	{attribute 'TcIecLibraryType'}
	{attribute 'external_name' := 'F_VN_RemapImageToPolarSpaceExp_GUID_737F4948_F24C_BB66_5AD3_96D65275813B'}
	(* Remap an image to polar space. (expert function) *)
	FUNCTION F_VN_RemapImageToPolarSpaceExp : HRESULT
	VAR_INPUT
		ipSrcImage	:	ITcVnImage;	(* Source image *)
		ipDestImage	:	REFERENCE TO ITcVnImage;	(* Destination image (Must not be the same as ipSrcImage! An appropriate destination image will be created if required.) *)
	END_VAR
	VAR_IN_OUT
		aCenter	:	TcVnPoint2_REAL;	(* Center point for the transformation *)
	END_VAR
	VAR_INPUT
		fMaxRadius	:	LREAL;	(* Maximum radius for the transformation (set to 0 for auto select) *)
		eInterpolationType	:	ETcVnInterpolationType;	(* Interpolation type *)
		hrPrev	:	HRESULT;	(* HRESULT indicating the result of previous operations (If SUCCEEDED(hrPrev) equals false, no operation is executed.) *)
	END_VAR

END_FUNCTION

// Functions/Geometric and Coordinate Transformations/F_VN_RemapImageToPolarSpaceExp2

	{attribute 'TcIecLibraryType'}
	{attribute 'external_name' := 'F_VN_RemapImageToPolarSpaceExp2_GUID_881403E3_891A_BA00_4A88_7979161734A7'}
	(* Remap an image to polar space. (expert function) *)
	FUNCTION F_VN_RemapImageToPolarSpaceExp2 : HRESULT
	VAR_INPUT
		ipSrcImage	:	ITcVnImage;	(* Source image *)
		ipDestImage	:	REFERENCE TO ITcVnImage;	(* Destination image (Must not be the same as ipSrcImage! An appropriate destination image will be created if required.) *)
	END_VAR
	VAR_IN_OUT
		aCenter	:	TcVnPoint2_REAL;	(* Center point for the transformation *)
	END_VAR
	VAR_INPUT
		fMaxRadius	:	LREAL;	(* Maximum radius for the transformation (set to 0 for auto select) *)
		eInterpolationType	:	ETcVnInterpolationType;	(* Interpolation type *)
		nDestWidth	:	DINT;	(* Destination image width (set to -1 for source image width, 0 to auto scale to transformed radius, > 0 for a user defined width) *)
		nDestHeight	:	DINT;	(* destination image height (set to -1 for source image height, 0 to auto scale to transformed radius * PI, > 0 for a user defined height) *)
		hrPrev	:	HRESULT;	(* HRESULT indicating the result of previous operations (If SUCCEEDED(hrPrev) equals false, no operation is executed.) *)
	END_VAR

END_FUNCTION

// Functions/Geometric and Coordinate Transformations/F_VN_ResizeImage

	{attribute 'TcIecLibraryType'}
	{attribute 'external_name' := 'F_VN_ResizeImage_GUID_066F6715_FDC4_B7AC_782D_C69A46C5F7F6'}
	(* Resize an image using a specific interpolation type. *)
	FUNCTION F_VN_ResizeImage : HRESULT
	VAR_INPUT
		ipSrcImage	:	ITcVnImage;	(* Source image *)
		ipDestImage	:	REFERENCE TO ITcVnImage;	(* Destination image (An appropriate image will be created if required.) *)
		nWidth	:	UDINT;	(* New width *)
		nHeight	:	UDINT;	(* New height *)
		eInterpolationType	:	ETcVnInterpolationType;	(* Interpolation type *)
		hrPrev	:	HRESULT;	(* HRESULT indicating the result of previous operations (If SUCCEEDED(hrPrev) equals false, no operation is executed.) *)
	END_VAR

END_FUNCTION

// Functions/Geometric and Coordinate Transformations/F_VN_ResizeImageExp

	{attribute 'TcIecLibraryType'}
	{attribute 'external_name' := 'F_VN_ResizeImageExp_GUID_DC68AAF5_744F_B632_6E74_ACED6F5A8BF2'}
	(* Resize an image using a specific interpolation type while maintaining its aspect ratio. (expert function) *)
	FUNCTION F_VN_ResizeImageExp : HRESULT
	VAR_INPUT
		ipSrcImage	:	ITcVnImage;	(* Source image *)
		ipDestImage	:	REFERENCE TO ITcVnImage;	(* Destination image (An appropriate image will be created if required.) *)
		nWidth	:	UDINT;	(* New width *)
		nHeight	:	UDINT;	(* New height *)
		eInterpolationType	:	ETcVnInterpolationType;	(* Interpolation type *)
		ePaddingMode	:	ETcVnPaddingMode;	(* Image padding mode *)
	END_VAR
	VAR_IN_OUT
		aBorderValue	:	TcVnVector4_LREAL;	(* Border value, if TCVN_PM_LETTERBOX is used *)
	END_VAR
	VAR_INPUT
		hrPrev	:	HRESULT;	(* HRESULT indicating the result of previous operations (If SUCCEEDED(hrPrev) equals false, no operation is executed.) *)
	END_VAR

END_FUNCTION

// Functions/Geometric and Coordinate Transformations/F_VN_RotateImage

	{attribute 'TcIecLibraryType'}
	{attribute 'external_name' := 'F_VN_RotateImage_GUID_67B496A2_F6DE_B78D_5711_982305E4D20B'}
	(* Rotate an image by 90, 180, or 270 degrees in clockwise direction. *)
	FUNCTION F_VN_RotateImage : HRESULT
	VAR_INPUT
		ipSrcImage	:	ITcVnImage;	(* Source image *)
		ipDestImage	:	REFERENCE TO ITcVnImage;	(* Destination image (An appropriate image will be created if required.) *)
		eAngle	:	ETcVnRotationAngle;	(* Rotation angle *)
		hrPrev	:	HRESULT;	(* HRESULT indicating the result of previous operations (If SUCCEEDED(hrPrev) equals false, no operation is executed.) *)
	END_VAR

END_FUNCTION

// Functions/Geometric and Coordinate Transformations/F_VN_RotateImageExp

	{attribute 'TcIecLibraryType'}
	{attribute 'external_name' := 'F_VN_RotateImageExp_GUID_493FD631_7649_B0AF_6E53_B79A69B64150'}
	(* Rotate an image by an individual rotation angle in degrees. *)
	FUNCTION F_VN_RotateImageExp : HRESULT
	VAR_INPUT
		ipSrcImage	:	ITcVnImage;	(* Source image *)
		ipDestImage	:	REFERENCE TO ITcVnImage;	(* Destination image (An appropriate image will be created if required.) *)
		fAngleDeg	:	LREAL;	(* Rotation angle in degree (positive: counter-clockwise, negative: clockwise) *)
		bAdjustDestSize	:	BOOL;	(* If true, ipDestImage size is adjusted so that the whole rotated ipSrcImage is contained. Otherwise, ipDestImage size is set to ipSrcImage size. *)
		hrPrev	:	HRESULT;	(* HRESULT indicating the result of previous operations (If SUCCEEDED(hrPrev) equals false, no operation is executed.) *)
	END_VAR

END_FUNCTION

// Functions/Geometric and Coordinate Transformations/F_VN_RotateImageExp2

	{attribute 'TcIecLibraryType'}
	{attribute 'external_name' := 'F_VN_RotateImageExp2_GUID_6EE8673E_D50E_BAEC_65C2_A62D1613988A'}
	(* Rotate an image by an individual rotation angle in degrees. (expert function) *)
	FUNCTION F_VN_RotateImageExp2 : HRESULT
	VAR_INPUT
		ipSrcImage	:	ITcVnImage;	(* Source image *)
		ipDestImage	:	REFERENCE TO ITcVnImage;	(* Destination image (An appropriate image will be created if required.) *)
		fAngleDeg	:	LREAL;	(* Rotation angle in degree (positive: counter-clockwise, negative: clockwise) *)
		bAdjustDestSize	:	BOOL;	(* If true, ipDestImage size is adjusted so that the whole rotated ipSrcImage is contained. Otherwise, ipDestImage size is set to ipSrcImage size. *)
		eInterpolationType	:	ETcVnInterpolationType;	(* Interpolation method *)
		eBorderInterpolation	:	ETcVnBorderInterpolationMethod;	(* Border interpolation method (ISOLATED not supported) *)
	END_VAR
	VAR_IN_OUT
		aBorderValue	:	TcVnVector4_LREAL;	(* Border value, if CONSTANT is used *)
	END_VAR
	VAR_INPUT
		hrPrev	:	HRESULT;	(* HRESULT indicating the result of previous operations (If SUCCEEDED(hrPrev) equals false, no operation is executed.) *)
	END_VAR

END_FUNCTION

// Functions/Geometric and Coordinate Transformations/F_VN_WarpAffineExp

	{attribute 'TcIecLibraryType'}
	{attribute 'external_name' := 'F_VN_WarpAffineExp_GUID_0ED46A98_6634_BCF0_4EEE_5250D0F0F4C5'}
	(* Apply an affine transformation to an image. (expert function) *)
	FUNCTION F_VN_WarpAffineExp : HRESULT
	VAR_INPUT
		ipSrcImage	:	ITcVnImage;	(* Source image *)
		ipDestImage	:	REFERENCE TO ITcVnImage;	(* Destination image (An appropriate image will be created if required.) *)
	END_VAR
	VAR_IN_OUT
		aTransformationMatrix	:	TcVnMatrix2x3_LREAL;	(* Affine transformation matrix *)
	END_VAR
	VAR_INPUT
		nDestWidth	:	UDINT;	(* Width of the destination image *)
		nDestHeight	:	UDINT;	(* Height of the destination image *)
		eInterpolationType	:	ETcVnInterpolationType;	(* Interpolation method *)
		bWarpInverse	:	BOOL;	(* Handle aTransformationMatrix as the inverse transformation *)
		eBorderInterpolation	:	ETcVnBorderInterpolationMethod;	(* Border interpolation method (ISOLATED not supported) *)
		fBorderValue	:	LREAL;	(* Border value, if CONSTANT is used *)
		hrPrev	:	HRESULT;	(* HRESULT indicating the result of previous operations (If SUCCEEDED(hrPrev) equals false, no operation is executed.) *)
	END_VAR

END_FUNCTION

// Functions/Geometric and Coordinate Transformations/F_VN_WarpAffine_Container

	{attribute 'TcIecLibraryType'}
	{attribute 'external_name' := 'F_VN_WarpAffine_Container_GUID_56BD7DA6_1D43_BE4D_7B12_DD5C0D5972CA'}
	(* Apply an affine transformation to a container of 2D points. *)
	FUNCTION F_VN_WarpAffine_Container : HRESULT
	VAR_INPUT
		ipSrcPoints	:	ITcVnContainer;	(* Source points (ContainerType_Vector_TcVnPoint2_DINT or ContainerType_Vector_TcVnPoint2_REAL or ContainerType_Vector_TcVnPoint2_LREAL) *)
		ipDestPoints	:	REFERENCE TO ITcVnContainer;	(* Returns the transformed points (same type ID as ipSrcPoints; Non-zero interface pointers are reused.) *)
	END_VAR
	VAR_IN_OUT
		aTransformationMatrix	:	TcVnMatrix2x3_LREAL;	(* Affine transformation matrix *)
	END_VAR
	VAR_INPUT
		hrPrev	:	HRESULT;	(* HRESULT indicating the result of previous operations (If SUCCEEDED(hrPrev) equals false, no operation is executed.) *)
	END_VAR

END_FUNCTION

// Functions/Geometric and Coordinate Transformations/F_VN_WarpAffine_Point

	{attribute 'TcIecLibraryType'}
	{attribute 'external_name' := 'F_VN_WarpAffine_Point_GUID_E77A0286_2158_BB35_4767_1C578A33A298'}
	(* Apply an affine transformation to a 2D point. *)
	FUNCTION F_VN_WarpAffine_Point : HRESULT
	VAR_IN_OUT
		aSrcPoint	:	TcVnPoint2_LREAL;	(* Source point *)
		aDestPoint	:	TcVnPoint2_LREAL;	(* Destination point *)
		aTransformationMatrix	:	TcVnMatrix2x3_LREAL;	(* Affine transformation matrix *)
	END_VAR
	VAR_INPUT
		hrPrev	:	HRESULT;	(* HRESULT indicating the result of previous operations (If SUCCEEDED(hrPrev) equals false, no operation is executed.) *)
	END_VAR

END_FUNCTION

// Functions/Geometric and Coordinate Transformations/F_VN_WarpAffine_Rectangle

	{attribute 'TcIecLibraryType'}
	{attribute 'external_name' := 'F_VN_WarpAffine_Rectangle_GUID_B71280DA_6C13_B846_4078_31BCF2965F61'}
	(* Use an affine transform to warp a rectangle. *)
	FUNCTION F_VN_WarpAffine_Rectangle : HRESULT
	VAR_INPUT
		nTopLeftX	:	UDINT;	(* x coordinate of the top left corner *)
		nTopLeftY	:	UDINT;	(* y coordinate of the top left corner *)
		nBottomRightX	:	UDINT;	(* x coordinate of the bottom right corner *)
		nBottomRightY	:	UDINT;	(* y coordinate of the bottom right corner *)
		ipDestPoints	:	REFERENCE TO ITcVnContainer;	(* Returns the 4 transformed points (ContainerType_Vector_TcVnPoint2_REAL) *)
	END_VAR
	VAR_IN_OUT
		aTransformationMatrix	:	TcVnMatrix2x3_LREAL;	(* Affine transformation matrix *)
	END_VAR
	VAR_INPUT
		hrPrev	:	HRESULT;	(* HRESULT indicating the result of previous operations (If SUCCEEDED(hrPrev) equals false, no operation is executed.) *)
	END_VAR

END_FUNCTION

// Functions/Geometric and Coordinate Transformations/F_VN_WarpPerspective

	{attribute 'TcIecLibraryType'}
	{attribute 'external_name' := 'F_VN_WarpPerspective_GUID_11483E27_169B_BD3A_571C_EBB12C538839'}
	(* Apply a perspective transformation to an image. *)
	FUNCTION F_VN_WarpPerspective : HRESULT
	VAR_INPUT
		ipSrcImage	:	ITcVnImage;	(* Source image *)
		ipDestImage	:	REFERENCE TO ITcVnImage;	(* Destination image (An appropriate image will be created if required.) *)
	END_VAR
	VAR_IN_OUT
		aTransformationMatrix	:	TcVnMatrix3x3_LREAL;	(* Perspective transformation matrix *)
	END_VAR
	VAR_INPUT
		hrPrev	:	HRESULT;	(* HRESULT indicating the result of previous operations (If SUCCEEDED(hrPrev) equals false, no operation is executed.) *)
	END_VAR

END_FUNCTION

// Functions/Geometric and Coordinate Transformations/F_VN_WarpPerspective_Container

	{attribute 'TcIecLibraryType'}
	{attribute 'external_name' := 'F_VN_WarpPerspective_Container_GUID_1A9D55A3_310D_B2CA_7120_BA66C8FDA0DB'}
	(* Apply a perspective transformation to a container of 2D points. *)
	FUNCTION F_VN_WarpPerspective_Container : HRESULT
	VAR_INPUT
		ipSrcPoints	:	ITcVnContainer;	(* Source points (ContainerType_Vector_TcVnPoint2_DINT or ContainerType_Vector_TcVnPoint2_REAL or ContainerType_Vector_TcVnPoint2_LREAL) *)
		ipDestPoints	:	REFERENCE TO ITcVnContainer;	(* Returns the transformed points (same type ID as ipSrcPoints; Non-zero interface pointers are reused.) *)
	END_VAR
	VAR_IN_OUT
		aTransformationMatrix	:	TcVnMatrix3x3_LREAL;	(* Perspective transformation matrix *)
	END_VAR
	VAR_INPUT
		hrPrev	:	HRESULT;	(* HRESULT indicating the result of previous operations (If SUCCEEDED(hrPrev) equals false, no operation is executed.) *)
	END_VAR

END_FUNCTION

// Functions/Geometric and Coordinate Transformations/F_VN_WarpPerspectiveExp

	{attribute 'TcIecLibraryType'}
	{attribute 'external_name' := 'F_VN_WarpPerspectiveExp_GUID_EA1E1C8D_C6BD_B82F_4255_245E461C95D7'}
	(* Apply a perspective transformation to an image. (expert function) *)
	FUNCTION F_VN_WarpPerspectiveExp : HRESULT
	VAR_INPUT
		ipSrcImage	:	ITcVnImage;	(* Source image *)
		ipDestImage	:	REFERENCE TO ITcVnImage;	(* Destination image (An appropriate image will be created if required.) *)
	END_VAR
	VAR_IN_OUT
		aTransformationMatrix	:	TcVnMatrix3x3_LREAL;	(* Perspective transformation matrix *)
	END_VAR
	VAR_INPUT
		nDestWidth	:	UDINT;	(* Width of the destination image *)
		nDestHeight	:	UDINT;	(* Height of the destination image *)
		eInterpolationType	:	ETcVnInterpolationType;	(* Interpolation method *)
		bWarpInverse	:	BOOL;	(* Handle aTransformationMatrix as the inverse transformation *)
		eBorderInterpolation	:	ETcVnBorderInterpolationMethod;	(* Border interpolation method (ISOLATED not supported) *)
		fBorderValue	:	LREAL;	(* Border value, if CONSTANT is used *)
		hrPrev	:	HRESULT;	(* HRESULT indicating the result of previous operations (If SUCCEEDED(hrPrev) equals false, no operation is executed.) *)
	END_VAR

END_FUNCTION

// Functions/Geometric and Coordinate Transformations/F_VN_WarpPerspective_Point

	{attribute 'TcIecLibraryType'}
	{attribute 'external_name' := 'F_VN_WarpPerspective_Point_GUID_E1C023CB_EEE0_BA8C_5D66_DED344D33911'}
	(* Apply a perspective transformation to a 2D point. *)
	FUNCTION F_VN_WarpPerspective_Point : HRESULT
	VAR_IN_OUT
		aSrcPoint	:	TcVnPoint2_LREAL;	(* Source point *)
		aDestPoint	:	TcVnPoint2_LREAL;	(* Destination point *)
		aTransformationMatrix	:	TcVnMatrix3x3_LREAL;	(* Perspective transformation matrix *)
	END_VAR
	VAR_INPUT
		hrPrev	:	HRESULT;	(* HRESULT indicating the result of previous operations (If SUCCEEDED(hrPrev) equals false, no operation is executed.) *)
	END_VAR

END_FUNCTION

// Functions/Geometric and Coordinate Transformations/F_VN_WarpPerspective_Rectangle

	{attribute 'TcIecLibraryType'}
	{attribute 'external_name' := 'F_VN_WarpPerspective_Rectangle_GUID_17AD1D40_0ED8_BEB6_46C5_9351EA5858B8'}
	(* Use a perspective transform to warp a rectangle. *)
	FUNCTION F_VN_WarpPerspective_Rectangle : HRESULT
	VAR_INPUT
		nTopLeftX	:	UDINT;	(* x coordinate of the top left corner *)
		nTopLeftY	:	UDINT;	(* y coordinate of the top left corner *)
		nBottomRightX	:	UDINT;	(* x coordinate of the bottom right corner *)
		nBottomRightY	:	UDINT;	(* y coordinate of the bottom right corner *)
		ipDestPoints	:	REFERENCE TO ITcVnContainer;	(* Returns the 4 transformed points (ContainerType_Vector_TcVnPoint2_REAL) *)
	END_VAR
	VAR_IN_OUT
		aTransformationMatrix	:	TcVnMatrix3x3_LREAL;	(* Perspective transformation matrix *)
	END_VAR
	VAR_INPUT
		hrPrev	:	HRESULT;	(* HRESULT indicating the result of previous operations (If SUCCEEDED(hrPrev) equals false, no operation is executed.) *)
	END_VAR

END_FUNCTION

// Functions/Image Color and Contrast Processing/F_VN_ApplyColorMap

	{attribute 'TcIecLibraryType'}
	{attribute 'external_name' := 'F_VN_ApplyColorMap_GUID_816CD833_E52B_BFA9_5F37_7447DD2AD7D0'}
	(* Apply a color map to a gray-level image. *)
	FUNCTION F_VN_ApplyColorMap : HRESULT
	VAR_INPUT
		ipSrcImage	:	ITcVnImage;	(* Source image (TCVN_ET_USINT or TCVN_ET_UINT, 1 channel) *)
		ipDestImage	:	REFERENCE TO ITcVnImage;	(* Returns the colored image (TCVN_ET_USINT, 3 channel. An appropriate image will be created if required.) *)
		ipColorMap	:	ITcVnContainer;	(* Color map to be applied to ipSrcImage (ContainerType_Vector_TcVnVector3_REAL with 256 or 65536 elements, dependent on ipSrcImage type). Can be either custom or created with F_VN_GenerateColorMap. *)
		hrPrev	:	HRESULT;	(* HRESULT indicating the result of previous operations (If SUCCEEDED(hrPrev) equals false, no operation is executed.) *)
	END_VAR

END_FUNCTION

// Functions/Image Color and Contrast Processing/F_VN_GenerateColorMap

	{attribute 'TcIecLibraryType'}
	{attribute 'external_name' := 'F_VN_GenerateColorMap_GUID_9FBF6773_DCEB_B6C6_7464_04D1C3DACD57'}
	(* Generates a pre-defined color map. *)
	FUNCTION F_VN_GenerateColorMap : HRESULT
	VAR_INPUT
		ipColorMap	:	REFERENCE TO ITcVnContainer;	(* Returns the color map (ContainerType_Vector_TcVnVector3_REAL with 256 or 65536 elements) *)
		eColorMap	:	ETcVnColorMap;	(* Selects a color map (similar to GNU Octave/MATLAB types) *)
		eColorMapSize	:	ETcVnColorMapSize;	(* Defines how many elements the generated color map should have *)
		hrPrev	:	HRESULT;	(* HRESULT indicating the result of previous operations (If SUCCEEDED(hrPrev) equals false, no operation is executed.) *)
	END_VAR

END_FUNCTION

// Functions/Image Color and Contrast Processing/F_VN_ApplyLut

	{attribute 'TcIecLibraryType'}
	{attribute 'external_name' := 'F_VN_ApplyLut_GUID_83DE5545_7633_BB82_50E7_190747D5A6CE'}
	(* Apply a lookup table to an image to manipulate its colors. *)
	FUNCTION F_VN_ApplyLut : HRESULT
	VAR_INPUT
		ipSrcImage	:	ITcVnImage;	(* Source image (1-4 channels of 8 or 16 bit types SINT, USINT, INT, UINT) *)
		ipDestImage	:	REFERENCE TO ITcVnImage;	(* Returns the result image (same size, type and channels as ipSrcImage. An appropriate image will be created if required.) *)
		ipLut	:	ITcVnContainer;	(* Lookup table with elements matching ipSrcImage type and either 256 (8 bit images) or 65536 (16 bit images) elements. E.g. ContainerType_Vector_USINT for 1-4 channel USINT image (in this case, the same lookup values are used for each channel) or ContainerType_Vector_TcVnVector3_USINT for a 3 channel USINT image (in this case, each channel uses an individual lookup value).
						 *)
		hrPrev	:	HRESULT;	(* HRESULT indicating the result of previous operations (If SUCCEEDED(hrPrev) equals false, no operation is executed.) *)
	END_VAR

END_FUNCTION

// Functions/Image Color and Contrast Processing/F_VN_Clahe

	{attribute 'TcIecLibraryType'}
	{attribute 'external_name' := 'F_VN_Clahe_GUID_B13FB575_AC4E_B224_67EF_0C730B48FF00'}
	(* Apply Constrast Limited Adaptive Histogram Equalization. This applies local histogram equalization to individual tiles. *)
	FUNCTION F_VN_Clahe : HRESULT
	VAR_INPUT
		ipSrcImage	:	ITcVnImage;	(* Source image (TCVN_ET_USINT or TCVN_ET_UINT, 1 channel) *)
		ipDestImage	:	REFERENCE TO ITcVnImage;	(* Returns the resulting image (An appropriate image will be created if required.) *)
		hrPrev	:	HRESULT;	(* HRESULT indicating the result of previous operations (If SUCCEEDED(hrPrev) equals false, no operation is executed.) *)
	END_VAR

END_FUNCTION

// Functions/Image Color and Contrast Processing/F_VN_ClaheExp

	{attribute 'TcIecLibraryType'}
	{attribute 'external_name' := 'F_VN_ClaheExp_GUID_0B0380D7_C764_B242_5B93_4C54EB94AC2E'}
	(* Apply Constrast Limited Adaptive Histogram Equalization. This applies local histogram equalization to individual tiles. (expert function) *)
	FUNCTION F_VN_ClaheExp : HRESULT
	VAR_INPUT
		ipSrcImage	:	ITcVnImage;	(* Source image (TCVN_ET_USINT or TCVN_ET_UINT, 1 channel) *)
		ipDestImage	:	REFERENCE TO ITcVnImage;	(* Returns the resulting image (An appropriate image will be created if required.) *)
		fClipLimit	:	LREAL;	(* Threshold for contrast limit (set to <= 0 to disable clipping) *)
		nTilesX	:	UDINT;	(* Number of tiles in x direction *)
		nTilesY	:	UDINT;	(* Number of tiles in y direction *)
		hrPrev	:	HRESULT;	(* HRESULT indicating the result of previous operations (If SUCCEEDED(hrPrev) equals false, no operation is executed.) *)
	END_VAR

END_FUNCTION

// Functions/Image Color and Contrast Processing/F_VN_ConvertColorSpace

	{attribute 'TcIecLibraryType'}
	{attribute 'external_name' := 'F_VN_ConvertColorSpace_GUID_E785C056_EC91_BB5D_5362_B1636F1941D4'}
	(* Convert image from one color space to another. *)
	FUNCTION F_VN_ConvertColorSpace : HRESULT
	VAR_INPUT
		ipSrcImage	:	ITcVnImage;	(* Source image *)
		ipDestImage	:	REFERENCE TO ITcVnImage;	(* Destination image (An appropriate destination image will be created if required.) *)
		eTransform	:	ETcVnColorSpaceTransform;	(* Transforms to be applied *)
		hrPrev	:	HRESULT;	(* HRESULT indicating the result of previous operations (If SUCCEEDED(hrPrev) equals false, no operation is executed.) *)
	END_VAR

END_FUNCTION

// Functions/Image Color and Contrast Processing/F_VN_GenerateCustomColorMap

	{attribute 'TcIecLibraryType'}
	{attribute 'external_name' := 'F_VN_GenerateCustomColorMap_GUID_FB8B79DD_6786_B6EC_65F8_CD6C6281E850'}
	(* Generate a custom color map by interpolating between user defined colors (equally distributed, linear for each channel). *)
	FUNCTION F_VN_GenerateCustomColorMap : HRESULT
	VAR_INPUT
		ipColorMap	:	REFERENCE TO ITcVnContainer;	(* Returns the color map (ContainerType_Vector_TcVnVector3_REAL with 256 or 65536 elements) *)
		ipInitialColors	:	ITcVnContainer;	(* User defined colors (ContainerType_Vector_TcVnVector3_REAL, at least 2 elements) *)
		eColorMapSize	:	ETcVnColorMapSize;	(* Defines how many elements the generated color map should have *)
		hrPrev	:	HRESULT;	(* HRESULT indicating the result of previous operations (If SUCCEEDED(hrPrev) equals false, no operation is executed.) *)
	END_VAR

END_FUNCTION

// Functions/Image Color and Contrast Processing/F_VN_Histogram

	{attribute 'TcIecLibraryType'}
	{attribute 'external_name' := 'F_VN_Histogram_GUID_97CA8631_C257_B622_4550_DD2D53C6AEF0'}
	(* Calculate the (multi-channel) histogram of an image. *)
	FUNCTION F_VN_Histogram : HRESULT
	VAR_INPUT
		ipSrcImage	:	ITcVnImage;	(* Source image *)
		ipDestHistogram	:	REFERENCE TO ITcVnContainer;	(* Returns a container with a multi-channel histogram, where every channel is represented as a vector of UDINT (ContainerType_Vector_Vector_UDINT. Non-zero interface pointers are reused.) *)
		hrPrev	:	HRESULT;	(* HRESULT indicating the result of previous operations (If SUCCEEDED(hrPrev) equals false, no operation is executed.) *)
	END_VAR

END_FUNCTION

// Functions/Image Color and Contrast Processing/F_VN_HistogramExp

	{attribute 'TcIecLibraryType'}
	{attribute 'external_name' := 'F_VN_HistogramExp_GUID_1CE0E788_2C38_B155_6387_B008436334A8'}
	(* Calculate the (multi-channel) histogram of an image. (expert function) *)
	FUNCTION F_VN_HistogramExp : HRESULT
	VAR_INPUT
		ipSrcImage	:	ITcVnImage;	(* Source image *)
		ipDestHistogram	:	REFERENCE TO ITcVnContainer;	(* Returns a container with a multi-channel histogram, where every channel is represented as a vector of UDINT (ContainerType_Vector_Vector_UDINT. Non-zero interface pointers are reused.) *)
	END_VAR
	VAR_IN_OUT
		nBins	:	UDINT;	(* Desired number of bins or 0 to keep the default for the corresponding image format (in) and default number of bins (out) *)
		fLowerBound	:	LREAL;	(* Lower (inclusive) boundary of the 0-th histogram bin (in), or receive the default if fLowerBound AND fUpperBound are set to 0 (out) *)
		fUpperBound	:	LREAL;	(* Upper (exclusive) boundary of the last histogram bin nBins-1 (in), or receive the default if fLowerBound AND fUpperBound are set to 0 (out) *)
	END_VAR
	VAR_INPUT
		ipMask	:	ITcVnImage;	(* Source image mask (TCVN_ET_USINT, 1 channel. Mask is optional, set to 0 if not required.) *)
		hrPrev	:	HRESULT;	(* HRESULT indicating the result of previous operations (If SUCCEEDED(hrPrev) equals false, no operation is executed.) *)
	END_VAR

END_FUNCTION

// Functions/Image Color and Contrast Processing/F_VN_HistogramEqualization

	{attribute 'TcIecLibraryType'}
	{attribute 'external_name' := 'F_VN_HistogramEqualization_GUID_3A0A3442_60A5_B388_5E3C_3DBC771CEFC5'}
	(* Equalize the histogram of a grayscale or rgb image, which normalizes the brightness and improves the contrast. *)
	FUNCTION F_VN_HistogramEqualization : HRESULT
	VAR_INPUT
		ipSrcImage	:	ITcVnImage;	(* Source image (USINT) *)
		ipDestImage	:	REFERENCE TO ITcVnImage;	(* Destination image (An appropriate destination image will be created if required.) *)
		hrPrev	:	HRESULT;	(* HRESULT indicating the result of previous operations (If SUCCEEDED(hrPrev) equals false, no operation is executed.) *)
	END_VAR

END_FUNCTION

// Functions/Image Color and Contrast Processing/F_VN_HistogramEqualizationExp

	{attribute 'TcIecLibraryType'}
	{attribute 'external_name' := 'F_VN_HistogramEqualizationExp_GUID_5019ED08_9A6E_BC80_7357_425A106A22F3'}
	(* Equalize the histogram of a grayscale or color image, which normalizes the brightness and improves the contrast. (expert function) 
	The channel index that should be equalized has to be specified (-1 expects a RGB image, converts it to YCbCr, equalizes the Y channel and converts the image back to RGB).  *)
	FUNCTION F_VN_HistogramEqualizationExp : HRESULT
	VAR_INPUT
		ipSrcImage	:	ITcVnImage;	(* Source image (USINT) *)
		ipDestImage	:	REFERENCE TO ITcVnImage;	(* Destination image (An appropriate destination image will be created if required.) *)
		nChannelIdx	:	INT;	(* Index of the image channel that should be equalized (-1 expects a RGB image, converts it to YCbCr, equalizes the Y channel and converts the image back to RGB) *)
		hrPrev	:	HRESULT;	(* HRESULT indicating the result of previous operations (If SUCCEEDED(hrPrev) equals false, no operation is executed.) *)
	END_VAR

END_FUNCTION

// Functions/Image Color and Contrast Processing/F_VN_InvertImageColor

	{attribute 'TcIecLibraryType'}
	{attribute 'external_name' := 'F_VN_InvertImageColor_GUID_E911183A_FFD5_BC4C_5076_3C639D48FDD8'}
	(* Invert the color of an image.
          For signed integer or negative floating point values, only the signs will be switched.
          If the image contains only positive floating point values, each pixel value is subtracted from the maximum available pixel value (or 1.0, whatever is higher). *)
	FUNCTION F_VN_InvertImageColor : HRESULT
	VAR_INPUT
		ipSrcImage	:	ITcVnImage;	(* Source image *)
		ipDestImage	:	REFERENCE TO ITcVnImage;	(* Destination image (An appropriate image will be created if required.) *)
		hrPrev	:	HRESULT;	(* HRESULT indicating the result of previous operations (If SUCCEEDED(hrPrev) equals false, no operation is executed.) *)
	END_VAR

END_FUNCTION

// Functions/Image Color and Contrast Processing/F_VN_InvertImageColorExp

	{attribute 'TcIecLibraryType'}
	{attribute 'external_name' := 'F_VN_InvertImageColorExp_GUID_06670B20_9EED_BCE6_6339_608C38CC3C14'}
	(* Invert the color of an image. (expert function)
          For signed integer or negative floating point values, only the signs will be switched.
          If the image contains only positive floating point values, each pixel value is subtracted from the maximum available pixel value (or 1.0, whatever is higher). *)
	FUNCTION F_VN_InvertImageColorExp : HRESULT
	VAR_INPUT
		ipSrcImage	:	ITcVnImage;	(* Source image *)
		ipDestImage	:	REFERENCE TO ITcVnImage;	(* Destination image (An appropriate image will be created if required.) *)
		fMaxValue	:	LREAL;	(* Maximum pixel value (e.g. if a 16 bit image contains 12 bit values). -1 means the default values are used. *)
		hrPrev	:	HRESULT;	(* HRESULT indicating the result of previous operations (If SUCCEEDED(hrPrev) equals false, no operation is executed.) *)
	END_VAR

END_FUNCTION

// Functions/Image Color and Contrast Processing/F_VN_NormalizeImage

	{attribute 'TcIecLibraryType'}
	{attribute 'external_name' := 'F_VN_NormalizeImage_GUID_DF64614F_1E7D_BDE6_6A3D_02BF884DF440'}
	(* Normalize an image regarding its value range (e.g. stretch pixel values [50..150] to full range [0..255]). *)
	FUNCTION F_VN_NormalizeImage : HRESULT
	VAR_INPUT
		ipSrcImage	:	ITcVnImage;	(* Source image *)
		ipDestImage	:	REFERENCE TO ITcVnImage;	(* Destination image (An appropriate destination image will be created if required.) *)
		hrPrev	:	HRESULT;	(* HRESULT indicating the result of previous operations (If SUCCEEDED(hrPrev) equals false, no operation is executed.) *)
	END_VAR

END_FUNCTION

// Functions/Image Color and Contrast Processing/F_VN_NormalizeImageExp

	{attribute 'TcIecLibraryType'}
	{attribute 'external_name' := 'F_VN_NormalizeImageExp_GUID_278826A3_5B31_B86C_4F2C_A4B2EC762E0C'}
	(* Normalize an image regarding its value range (e.g. stretch pixel values [50..150] to full range [0..255]) or scale the values regarding a specific normalization (e.g. L2-norm). (expert function) *)
	FUNCTION F_VN_NormalizeImageExp : HRESULT
	VAR_INPUT
		ipSrcImage	:	ITcVnImage;	(* Source image *)
		ipDestImage	:	REFERENCE TO ITcVnImage;	(* Destination image (An appropriate destination image will be created if required.) *)
		fAlpha	:	LREAL;	(* Lower range boundary (in case of normalizing the value range) or value to normalize to (||ipDestImage|| = fAlpha) *)
		fBeta	:	LREAL;	(* Upper range boundary (in case of normalizing the value range) *)
		eNormType	:	ETcVnNormalizationType;	(* Normalization type (only INF, L1, L2 or MINMAX) *)
		eDestType	:	ETcVnElementType;	(* Destination image depth (usually SAME_AS_SOURCE) *)
		ipMask	:	ITcVnImage;	(* Mask to restrict the normalization to specific pixel positions (set 0 to normalize the whole image) *)
		hrPrev	:	HRESULT;	(* HRESULT indicating the result of previous operations (If SUCCEEDED(hrPrev) equals false, no operation is executed.) *)
	END_VAR

END_FUNCTION

// Functions/Image Color and Contrast Processing/F_VN_NormalizeImageForDisplay

	{attribute 'TcIecLibraryType'}
	{attribute 'external_name' := 'F_VN_NormalizeImageForDisplay_GUID_849482CC_D1BF_B1BB_6D8E_6AC161F307DE'}
	(* Normalize an image for display, i.e. scale it to the full value range of the underlying data type (-1 to 1 for floating point). *)
	FUNCTION F_VN_NormalizeImageForDisplay : HRESULT
	VAR_INPUT
		ipSrcImage	:	ITcVnImage;	(* Source image *)
		ipDestImage	:	REFERENCE TO ITcVnImage;	(* Destination image (An appropriate destination image will be created if required.) *)
		eSignedNormalization	:	ETcVnSignedNormalization;	(* Option for normalizing signed values *)
		hrPrev	:	HRESULT;	(* HRESULT indicating the result of previous operations (If SUCCEEDED(hrPrev) equals false, no operation is executed.) *)
	END_VAR

END_FUNCTION

// Functions/Image Color and Contrast Processing/F_VN_ReferenceColorSimilarity_ITcVnColorModel

	{attribute 'TcIecLibraryType'}
	{attribute 'external_name' := 'F_VN_ReferenceColorSimilarity_ITcVnColorModel_GUID_F4B25797_7917_B8FC_5558_54102443F353'}
	(* Computes the similarity to a reference color model for each pixel in the source image. *)
	FUNCTION F_VN_ReferenceColorSimilarity_ITcVnColorModel : HRESULT
	VAR_INPUT
		ipSrcImage	:	ITcVnImage;	(* RGB source image (USINT, 3 channels) *)
		ipDestImage	:	REFERENCE TO ITcVnImage;	(* Returns the similarity to ipColorModel for each pixel in ipSrcImage (USINT, 1 channel. An appropriate destination image will be created if required.) *)
		ipColorModel	:	ITcVnColorModel;	(* Color model *)
		hrPrev	:	HRESULT;	(* HRESULT indicating the result of previous operations (If SUCCEEDED(hrPrev) equals false, no operation is executed.) *)
	END_VAR

END_FUNCTION

// Interfaces/Machine Learning/ITcVnColorModel

	(* Interface to train and classify an image color. *)
	{attribute 'c++_compatible'}
	{attribute 'vtable_order' := 'TrainImageColor;ClassifyImageColor'}
	INTERFACE ITcVnColorModel EXTENDS ITcVnMlModel


(* Train the color of the provided image. *)
	{attribute 'c++_compatible'}
	{attribute 'minimal_input_size' := '4'}
	{attribute 'pack_mode' := '4'}
	METHOD TrainImageColor : HRESULT
	VAR_INPUT
		ipSrcImage : ITcVnImage;
		nDifferentColors : UDINT;
		ipMask : ITcVnImage;
		nSkipPixels : UDINT;
	END_VAR
END_METHOD


(* Compute the similarity of each image pixel to the trained reference color. *)
	{attribute 'c++_compatible'}
	{attribute 'minimal_input_size' := '4'}
	{attribute 'pack_mode' := '4'}
	METHOD ClassifyImageColor : HRESULT
	VAR_INPUT
		ipSrcImage : ITcVnImage;
		pipDestImage : POINTER TO ITcVnImage;
		fVariance : REAL;
		fLuminanceWeight : REAL;
	END_VAR
END_METHOD

END_INTERFACE

// Functions/Image Color and Contrast Processing/F_VN_ReferenceColorSimilarityExp_ITcVnColorModel

	{attribute 'TcIecLibraryType'}
	{attribute 'external_name' := 'F_VN_ReferenceColorSimilarityExp_ITcVnColorModel_GUID_F0AE672C_F0E6_B94B_7FE1_8AB59959B227'}
	(* Computes the similarity to a reference color model for each pixel in the source image. (expert function) *)
	FUNCTION F_VN_ReferenceColorSimilarityExp_ITcVnColorModel : HRESULT
	VAR_INPUT
		ipSrcImage	:	ITcVnImage;	(* RGB source image (USINT, 3 channels) *)
		ipDestImage	:	REFERENCE TO ITcVnImage;	(* Returns the similarity to ipColorModel for each pixel in ipSrcImage (USINT, 1 channel. An appropriate destination image will be created if required.) *)
		ipColorModel	:	ITcVnColorModel;	(* Color model *)
		fVariance	:	REAL;	(* Allowed color variance (0.1 - 0.3 might be a good start to try) *)
		fLuminanceWeight	:	REAL;	(* Weight the impact of the luminance ([0..1], e.g. set to 0 to be more resistant to unequal illumination, but might be required to differentiate between some colors. Ignored if ipColorModel is of type RGB.) *)
		hrPrev	:	HRESULT;	(* HRESULT indicating the result of previous operations (If SUCCEEDED(hrPrev) equals false, no operation is executed.) *)
	END_VAR

END_FUNCTION

// Functions/Image Color and Contrast Processing/F_VN_ReferenceColorSimilarity_ITcVnMlModel

	{attribute 'TcIecLibraryType'}
	{attribute 'external_name' := 'F_VN_ReferenceColorSimilarity_ITcVnMlModel_GUID_A4DF2C39_3B8B_B7CE_623E_B2233126C047'}
	(* Computes the similarity to a reference color model for each pixel in the source image. *)
	FUNCTION F_VN_ReferenceColorSimilarity_ITcVnMlModel : HRESULT
	VAR_INPUT
		ipSrcImage	:	ITcVnImage;	(* RGB source image (USINT, 3 channels) *)
		ipDestImage	:	REFERENCE TO ITcVnImage;	(* Returns the similarity to ipColorModel for each pixel in ipSrcImage (USINT, 1 channel. An appropriate destination image will be created if required.) *)
		ipColorModel	:	ITcVnMlModel;	(* Color model *)
		hrPrev	:	HRESULT;	(* HRESULT indicating the result of previous operations (If SUCCEEDED(hrPrev) equals false, no operation is executed.) *)
	END_VAR

END_FUNCTION

// Functions/Image Color and Contrast Processing/F_VN_ReferenceColorSimilarityExp_ITcVnMlModel

	{attribute 'TcIecLibraryType'}
	{attribute 'external_name' := 'F_VN_ReferenceColorSimilarityExp_ITcVnMlModel_GUID_8603549B_3D85_B25B_5257_608AC1C84E02'}
	(* Computes the similarity to a reference color model for each pixel in the source image. (expert function) *)
	FUNCTION F_VN_ReferenceColorSimilarityExp_ITcVnMlModel : HRESULT
	VAR_INPUT
		ipSrcImage	:	ITcVnImage;	(* RGB source image (USINT, 3 channels) *)
		ipDestImage	:	REFERENCE TO ITcVnImage;	(* Returns the similarity to ipColorModel for each pixel in ipSrcImage (USINT, 1 channel. An appropriate destination image will be created if required.) *)
		ipColorModel	:	ITcVnMlModel;	(* Color model *)
		fVariance	:	REAL;	(* Allowed color variance (0.1 - 0.3 might be a good start to try) *)
		fLuminanceWeight	:	REAL;	(* Weight the impact of the luminance ([0..1], e.g. set to 0 to be more resistant to unequal illumination, but might be required to differentiate between some colors. Ignored if ipColorModel is of type RGB.) *)
		hrPrev	:	HRESULT;	(* HRESULT indicating the result of previous operations (If SUCCEEDED(hrPrev) equals false, no operation is executed.) *)
	END_VAR

END_FUNCTION

// Functions/Image Color and Contrast Processing/F_VN_ReferenceColorSimilarity_TcVnVector3_LREAL

	{attribute 'TcIecLibraryType'}
	{attribute 'external_name' := 'F_VN_ReferenceColorSimilarity_TcVnVector3_LREAL_GUID_2452A6E4_481B_B108_6A9D_A006EDDB667C'}
	(* Computes the similarity to a reference color for each pixel in the source image. *)
	FUNCTION F_VN_ReferenceColorSimilarity_TcVnVector3_LREAL : HRESULT
	VAR_INPUT
		ipSrcImage	:	ITcVnImage;	(* RGB source image (USINT, 3 channels) *)
		ipDestImage	:	REFERENCE TO ITcVnImage;	(* Returns the similarity to aRefColor for each pixel in ipSrcImage (USINT, 1 channel. An appropriate destination image will be created if required.) *)
	END_VAR
	VAR_IN_OUT
		aRefColor	:	TcVnVector3_LREAL;	(* Reference color (RGB, [0..255]) *)
	END_VAR
	VAR_INPUT
		hrPrev	:	HRESULT;	(* HRESULT indicating the result of previous operations (If SUCCEEDED(hrPrev) equals false, no operation is executed.) *)
	END_VAR

END_FUNCTION

// Functions/Image Color and Contrast Processing/F_VN_ReferenceColorSimilarityExp_TcVnVector3_LREAL

	{attribute 'TcIecLibraryType'}
	{attribute 'external_name' := 'F_VN_ReferenceColorSimilarityExp_TcVnVector3_LREAL_GUID_0DD98DE1_6BFD_BBDD_5E45_F31504BAFE68'}
	(* Computes the similarity to a reference color for each pixel in the source image. (expert function) *)
	FUNCTION F_VN_ReferenceColorSimilarityExp_TcVnVector3_LREAL : HRESULT
	VAR_INPUT
		ipSrcImage	:	ITcVnImage;	(* RGB source image (USINT, 3 channels) *)
		ipDestImage	:	REFERENCE TO ITcVnImage;	(* Returns the similarity to aRefColor for each pixel in ipSrcImage (USINT, 1 channel. An appropriate destination image will be created if required.) *)
	END_VAR
	VAR_IN_OUT
		aRefColor	:	TcVnVector3_LREAL;	(* Reference color (RGB, [0..255]) *)
	END_VAR
	VAR_INPUT
		fVariance	:	REAL;	(* Allowed color variance (0.1 - 0.3 might be a good start to try) *)
		fLuminanceWeight	:	REAL;	(* Weight the impact of the luminance ([0..1], e.g. set to 0 to be more resistant to unequal illumination, but might be required to differentiate between some colors) *)
		hrPrev	:	HRESULT;	(* HRESULT indicating the result of previous operations (If SUCCEEDED(hrPrev) equals false, no operation is executed.) *)
	END_VAR

END_FUNCTION

// Functions/Image Color and Contrast Processing/F_VN_TrainImageColor

	{attribute 'TcIecLibraryType'}
	{attribute 'external_name' := 'F_VN_TrainImageColor_GUID_DC2BFB0F_4E1B_B195_5ECB_7BE6866D18CC'}
	(* Create a new color model, describing the image color. *)
	FUNCTION F_VN_TrainImageColor : HRESULT
	VAR_INPUT
		ipSrcImage	:	ITcVnImage;	(* Source image (3 channels (RGB) of type USINT) *)
		ipColorModel	:	REFERENCE TO ITcVnColorModel;	(* Returns the color model *)
		nDifferentColors	:	UDINT;	(* Number of different colors to distinguish *)
		hrPrev	:	HRESULT;	(* HRESULT indicating the result of previous operations (If SUCCEEDED(hrPrev) equals false, no operation is executed.) *)
	END_VAR

END_FUNCTION

// Functions/Image Color and Contrast Processing/F_VN_TrainImageColorExp

	{attribute 'TcIecLibraryType'}
	{attribute 'external_name' := 'F_VN_TrainImageColorExp_GUID_BFFE78A6_D5B8_B6E7_79D5_27A05FC83135'}
	(* Create a new color model, describing the image color. (expert function) *)
	FUNCTION F_VN_TrainImageColorExp : HRESULT
	VAR_INPUT
		ipSrcImage	:	ITcVnImage;	(* Source image (3 channels (RGB) of type USINT) *)
		ipColorModel	:	REFERENCE TO ITcVnColorModel;	(* Returns the color model *)
		nDifferentColors	:	UDINT;	(* Number of different colors to distinguish *)
		eMethod	:	ETcVnColorTrainingMethod;	(* Color training method *)
		ipMask	:	ITcVnImage;	(* Optional image mask (1 channel of type USINT, set to 0 if not required) *)
		nSkipPixels	:	UDINT;	(* Number of pixels to skip between each evaluated color sample (to achieve a better performance). 0 takes every pixel into account and tends to be more accurate. *)
		hrPrev	:	HRESULT;	(* HRESULT indicating the result of previous operations (If SUCCEEDED(hrPrev) equals false, no operation is executed.) *)
	END_VAR

END_FUNCTION

// Functions/Image Color and Contrast Processing/F_VN_TrainImageColorExp2

	{attribute 'TcIecLibraryType'}
	{attribute 'external_name' := 'F_VN_TrainImageColorExp2_GUID_DACF3D5F_DD5E_BE45_6BA2_5AEAE7495463'}
	(* Create a new color model, describing the image color. (expert function) *)
	FUNCTION F_VN_TrainImageColorExp2 : HRESULT
	VAR_INPUT
		ipSrcImage	:	ITcVnImage;	(* Source image (3 channels (RGB) of type USINT) *)
		ipColorModel	:	REFERENCE TO ITcVnColorModel;	(* Returns the color model *)
		nDifferentColors	:	UDINT;	(* Maximum number of different colors to distinguish (if LBG is used as a clustering algorithm, the result might have less different colors, depending on nMaxClusterRadius) *)
		eMethod	:	ETcVnColorTrainingMethod;	(* Color training method *)
		ipMask	:	ITcVnImage;	(* Optional image mask (1 channel of type USINT, set to 0 if not required) *)
		nSkipPixels	:	UDINT;	(* Number of pixels to skip between each evaluated color sample (to achieve a better performance). 0 takes every pixel into account and tends to be more accurate. *)
		eClusteringAlgorithm	:	ETcVnClusteringAlgorithm;	(* Clustering algorithm *)
		nMaxClusterRadius	:	DINT;	(* Only used for the LBG clustering algorithm. Maximum allowed radius (> 0) of a single cluster, i.e. clusters with a higher radius will be split into smaller ones, until a global number of nDifferentColors is reached. *)
		bSingleSplitSteps	:	BOOL;	(* Only used for the LBG clustering algorithm. If true, the global optimization is always run after a single cluster has been split. If false, several clusters are split within the same step before applying the global optimization. Applying the global optimization less often is faster, but can lead to less optimal results, especially having 2 nearby clusters that could be represented by 1) *)
		hrPrev	:	HRESULT;	(* HRESULT indicating the result of previous operations (If SUCCEEDED(hrPrev) equals false, no operation is executed.) *)
	END_VAR

END_FUNCTION

// Functions/Image Color and Contrast Processing/F_VN_TrainImageColor_ITcVnMlModel

	{attribute 'TcIecLibraryType'}
	{attribute 'external_name' := 'F_VN_TrainImageColor_ITcVnMlModel_GUID_9728FB0F_CD18_B61F_6CE1_38DBE22EA6CB'}
	(* Create a new color model, describing the image color. *)
	FUNCTION F_VN_TrainImageColor_ITcVnMlModel : HRESULT
	VAR_INPUT
		ipSrcImage	:	ITcVnImage;	(* Source image (3 channels (RGB) of type USINT) *)
		ipColorModel	:	REFERENCE TO ITcVnMlModel;	(* Returns the color model *)
		nDifferentColors	:	UDINT;	(* Number of different colors to distinguish *)
		hrPrev	:	HRESULT;	(* HRESULT indicating the result of previous operations (If SUCCEEDED(hrPrev) equals false, no operation is executed.) *)
	END_VAR

END_FUNCTION

// Functions/Image Color and Contrast Processing/F_VN_TrainImageColorExp_ITcVnMlModel

	{attribute 'TcIecLibraryType'}
	{attribute 'external_name' := 'F_VN_TrainImageColorExp_ITcVnMlModel_GUID_34C68F01_8251_B48B_53F2_921840517D35'}
	(* Create a new color model, describing the image color. (expert function) *)
	FUNCTION F_VN_TrainImageColorExp_ITcVnMlModel : HRESULT
	VAR_INPUT
		ipSrcImage	:	ITcVnImage;	(* Source image (3 channels (RGB) of type USINT) *)
		ipColorModel	:	REFERENCE TO ITcVnMlModel;	(* Returns the color model *)
		nDifferentColors	:	UDINT;	(* Number of different colors to distinguish *)
		eMethod	:	ETcVnColorTrainingMethod;	(* Color training method *)
		ipMask	:	ITcVnImage;	(* Optional image mask (1 channel of type USINT, set to 0 if not required) *)
		nSkipPixels	:	UDINT;	(* Number of pixels to skip between each evaluated color sample (to achieve a better performance). 0 takes every pixel into account and tends to be more accurate. *)
		hrPrev	:	HRESULT;	(* HRESULT indicating the result of previous operations (If SUCCEEDED(hrPrev) equals false, no operation is executed.) *)
	END_VAR

END_FUNCTION

// Functions/Image Color and Contrast Processing/F_VN_TrainImageColorExp2_ITcVnMlModel

	{attribute 'TcIecLibraryType'}
	{attribute 'external_name' := 'F_VN_TrainImageColorExp2_ITcVnMlModel_GUID_8CFC34DA_2EA5_BC5E_602F_A37085D7DC82'}
	(* Create a new color model, describing the image color. (expert function) *)
	FUNCTION F_VN_TrainImageColorExp2_ITcVnMlModel : HRESULT
	VAR_INPUT
		ipSrcImage	:	ITcVnImage;	(* Source image (3 channels (RGB) of type USINT) *)
		ipColorModel	:	REFERENCE TO ITcVnMlModel;	(* Returns the color model *)
		nDifferentColors	:	UDINT;	(* Maximum number of different colors to distinguish (if LBG is used as a clustering algorithm, the result might have less different colors, depending on nMaxClusterRadius) *)
		eMethod	:	ETcVnColorTrainingMethod;	(* Color training method *)
		ipMask	:	ITcVnImage;	(* Optional image mask (1 channel of type USINT, set to 0 if not required) *)
		nSkipPixels	:	UDINT;	(* Number of pixels to skip between each evaluated color sample (to achieve a better performance). 0 takes every pixel into account and tends to be more accurate. *)
		eClusteringAlgorithm	:	ETcVnClusteringAlgorithm;	(* Clustering algorithm *)
		nMaxClusterRadius	:	DINT;	(* Only used for the LBG clustering algorithm. Maximum allowed radius (> 0) of a single cluster, i.e. clusters with a higher radius will be split into smaller ones, until a global number of nDifferentColors is reached. *)
		bSingleSplitSteps	:	BOOL;	(* Only used for the LBG clustering algorithm. If true, the global optimization is always run after a single cluster has been split. If false, several clusters are split within the same step before applying the global optimization. Applying the global optimization less often is faster, but can lead to less optimal results, especially having 2 nearby clusters that could be represented by 1) *)
		hrPrev	:	HRESULT;	(* HRESULT indicating the result of previous operations (If SUCCEEDED(hrPrev) equals false, no operation is executed.) *)
	END_VAR

END_FUNCTION

// Functions/Image Color and Contrast Processing/F_VN_WhiteBalance

	{attribute 'TcIecLibraryType'}
	{attribute 'external_name' := 'F_VN_WhiteBalance_GUID_44ADDC56_8B35_BE2F_4CAB_A0C50204933D'}
	(* Calculates the white balance ratios for a RGB image. Uses the green channel as a reference and computes the relative ratios for the red and blue channels. Requires a non-reflecting, not overexposed white colored object (e.g. a sheet of paper) in at least 100 pixels of the image to provide reasonable results. The resulting ratios can then be set on the camera (multiply with existing ratios), or applied in the PLC via MultiplyImageWithVector. *)
	FUNCTION F_VN_WhiteBalance : HRESULT
	VAR_INPUT
		ipSrcImage	:	ITcVnImage;	(* Source image (3 channels (RGB), USINT or UINT) *)
		ipDestImage	:	REFERENCE TO ITcVnImage;	(* Destination image with white balance applied (optional, set to 0 if not required. An appropriate image will be created if required.) *)
		fRatioRed	:	REFERENCE TO REAL;	(* Returns the ratio for the red channel *)
		fRatioBlue	:	REFERENCE TO REAL;	(* Returns the ratio for the blue channel *)
		nMaxValue	:	UDINT;	(* Specify the maximum pixel value that would be achieved by overexposure (usually 255 for 8 bit or 4095 for 12 bit data) *)
		hrPrev	:	HRESULT;	(* HRESULT indicating the result of previous operations (If SUCCEEDED(hrPrev) equals false, no operation is executed.) *)
	END_VAR

END_FUNCTION

// Functions/Contour Analysis/F_VN_ApproximatePolygon

	{attribute 'TcIecLibraryType'}
	{attribute 'external_name' := 'F_VN_ApproximatePolygon_GUID_78D8B309_B69B_B3C9_648E_967EFCC9C3CD'}
	(* Approximate a contour to a simplified polygon (using the Douglas-Peucker algorithm). *)
	FUNCTION F_VN_ApproximatePolygon : HRESULT
	VAR_INPUT
		ipSrcContour	:	ITcVnContainer;	(* Single contour (ContainerType_Vector_TcVnPoint2_DINT or ContainerType_Vector_TcVnPoint2_REAL; The elements of this container are the points of the contour.) *)
		ipDestContour	:	REFERENCE TO ITcVnContainer;	(* Returns a container which is filled with the approximated polygon points (same type ID as ipSrcContour; Non-zero interface pointers are reused.) *)
		fMaxDist	:	LREAL;	(* Maximum distance between the original contour and its approximation *)
		bClosed	:	BOOL;	(* Specify, if the contour is closed (first and last points connected) or not *)
		hrPrev	:	HRESULT;	(* HRESULT indicating the result of previous operations (If SUCCEEDED(hrPrev) equals false, no operation is executed.) *)
	END_VAR

END_FUNCTION

// Functions/Contour Analysis/F_VN_CheckIfPointIsInsideContour

	{attribute 'TcIecLibraryType'}
	{attribute 'external_name' := 'F_VN_CheckIfPointIsInsideContour_GUID_BDDDB352_B1EE_BDA2_7893_7A957C9DC97F'}
	(* Checks if a point is inside a contour (and optionally return the distance to it). *)
	FUNCTION F_VN_CheckIfPointIsInsideContour : HRESULT
	VAR_INPUT
		ipContour	:	ITcVnContainer;	(* Single contour (ContainerType_Vector_TcVnPoint2_DINT or ContainerType_Vector_TcVnPoint2_REAL) *)
	END_VAR
	VAR_IN_OUT
		aPoint	:	TcVnPoint2_REAL;	(* Point position to check *)
		fDist	:	LREAL;	(* Returns the result (> 0: the point is inside the contour; 0: the point is on the contour; < 0: the point is outside the contour) *)
	END_VAR
	VAR_INPUT
		bMeasureDistance	:	BOOL;	(* If true, fDist returns the distance to the nearest contour edge. Otherwise, fDist only returns -1, 0 or +1 (recommended to set to false if the distance is not required, as this is faster). *)
		hrPrev	:	HRESULT;	(* HRESULT indicating the result of previous operations (If SUCCEEDED(hrPrev) equals false, no operation is executed.) *)
	END_VAR

END_FUNCTION

// Functions/Contour Analysis/F_VN_ContourArea

	{attribute 'TcIecLibraryType'}
	{attribute 'external_name' := 'F_VN_ContourArea_GUID_6C17E99B_3463_B4AC_5256_2009ADDF76E1'}
	(* Estimate the contour area using Green's formula. *)
	FUNCTION F_VN_ContourArea : HRESULT
	VAR_INPUT
		ipContour	:	ITcVnContainer;	(* Single contour (ContainerType_Vector_TcVnPoint2_DINT or ContainerType_Vector_TcVnPoint2_REAL; The elements of this container are the points of the contour.) *)
	END_VAR
	VAR_IN_OUT
		fArea	:	LREAL;	(* Returns the estimated contour area (The actual contour area may differ depending on the shape of the contour.) *)
	END_VAR
	VAR_INPUT
		hrPrev	:	HRESULT;	(* HRESULT indicating the result of previous operations (If SUCCEEDED(hrPrev) equals false, no operation is executed.) *)
	END_VAR

END_FUNCTION

// Functions/Contour Analysis/F_VN_ContourCenterOfMass

	{attribute 'TcIecLibraryType'}
	{attribute 'external_name' := 'F_VN_ContourCenterOfMass_GUID_D073B3CA_9036_B053_451F_D6EA301F31DC'}
	(* Computes the center of mass of a contour. *)
	FUNCTION F_VN_ContourCenterOfMass : HRESULT
	VAR_INPUT
		ipContour	:	ITcVnContainer;	(* Single contour (ContainerType_Vector_TcVnPoint2_DINT or ContainerType_Vector_TcVnPoint2_REAL; The elements of this container are the points of the contour.) *)
	END_VAR
	VAR_IN_OUT
		aCenterOfMass	:	TcVnPoint2_LREAL;	(* Returns the center of mass of the contour *)
	END_VAR
	VAR_INPUT
		hrPrev	:	HRESULT;	(* HRESULT indicating the result of previous operations (If SUCCEEDED(hrPrev) equals false, no operation is executed.) *)
	END_VAR

END_FUNCTION

// Functions/Contour Analysis/F_VN_ContourCircularity

	{attribute 'TcIecLibraryType'}
	{attribute 'external_name' := 'F_VN_ContourCircularity_GUID_2A9805CD_95B1_B899_4BC7_D5AA7C7453FA'}
	(* Computes the circularity of a contour (1.0: ideal circle, 0.0: straight line). *)
	FUNCTION F_VN_ContourCircularity : HRESULT
	VAR_INPUT
		ipContour	:	ITcVnContainer;	(* Single contour (ContainerType_Vector_TcVnPoint2_DINT or ContainerType_Vector_TcVnPoint2_REAL; The elements of this container are the points of the contour.) *)
	END_VAR
	VAR_IN_OUT
		fCircularity	:	LREAL;	(* Returns the circularity of the contour [0..1] *)
	END_VAR
	VAR_INPUT
		hrPrev	:	HRESULT;	(* HRESULT indicating the result of previous operations (If SUCCEEDED(hrPrev) equals false, no operation is executed.) *)
	END_VAR

END_FUNCTION

// Functions/Contour Analysis/F_VN_ContourConvexity

	{attribute 'TcIecLibraryType'}
	{attribute 'external_name' := 'F_VN_ContourConvexity_GUID_C4F69F8C_B238_BF1A_6D61_D3DD5C72D3B1'}
	(* Computes the convexity of a contour as the ratio between the contour's area and the area of the convex hull (1.0: convex shapes (i.e. rectangle, circle, ..., etc.), 0.0: zero area (i.e. a line or an empty contour)). *)
	FUNCTION F_VN_ContourConvexity : HRESULT
	VAR_INPUT
		ipContour	:	ITcVnContainer;	(* Single contour (ContainerType_Vector_TcVnPoint2_DINT or ContainerType_Vector_TcVnPoint2_REAL; The elements of this container are the points of the contour.) *)
	END_VAR
	VAR_IN_OUT
		fConvexity	:	LREAL;	(* Returns the convexity of the contour [0..1] *)
	END_VAR
	VAR_INPUT
		hrPrev	:	HRESULT;	(* HRESULT indicating the result of previous operations (If SUCCEEDED(hrPrev) equals false, no operation is executed.) *)
	END_VAR

END_FUNCTION

// Functions/Contour Analysis/F_VN_ContourEccentricity

	{attribute 'TcIecLibraryType'}
	{attribute 'external_name' := 'F_VN_ContourEccentricity_GUID_4B2A9822_603F_B1D8_67EB_7C4EAE8E9630'}
	(* Computes the eccentricity of a contour (0.0: circular, 1.0: linear). *)
	FUNCTION F_VN_ContourEccentricity : HRESULT
	VAR_INPUT
		ipContour	:	ITcVnContainer;	(* Single contour (ContainerType_Vector_TcVnPoint2_DINT or ContainerType_Vector_TcVnPoint2_REAL; The elements of this container are the points of the contour.) *)
	END_VAR
	VAR_IN_OUT
		fEccentricity	:	LREAL;	(* Returns the eccentricity of the contour [0..1] *)
	END_VAR
	VAR_INPUT
		hrPrev	:	HRESULT;	(* HRESULT indicating the result of previous operations (If SUCCEEDED(hrPrev) equals false, no operation is executed.) *)
	END_VAR

END_FUNCTION

// Functions/Contour Analysis/F_VN_ContourElongation

	{attribute 'TcIecLibraryType'}
	{attribute 'external_name' := 'F_VN_ContourElongation_GUID_E62D0B81_BC4F_B73B_61F0_4BC5534B22CC'}
	(* Computes the elongation factor of a contour. *)
	FUNCTION F_VN_ContourElongation : HRESULT
	VAR_INPUT
		ipContour	:	ITcVnContainer;	(* Single contour (ContainerType_Vector_TcVnPoint2_DINT or ContainerType_Vector_TcVnPoint2_REAL; The elements of this container are the points of the contour.) *)
	END_VAR
	VAR_IN_OUT
		fElongation	:	LREAL;	(* Returns the elongation of the contour *)
	END_VAR
	VAR_INPUT
		hrPrev	:	HRESULT;	(* HRESULT indicating the result of previous operations (If SUCCEEDED(hrPrev) equals false, no operation is executed.) *)
	END_VAR

END_FUNCTION

// Functions/Contour Analysis/F_VN_ContourExtremePoint

	{attribute 'TcIecLibraryType'}
	{attribute 'external_name' := 'F_VN_ContourExtremePoint_GUID_3B8E8AEE_8647_BE9F_6ADA_672DA220841B'}
	(* Finds the contour extreme point. *)
	FUNCTION F_VN_ContourExtremePoint : HRESULT
	VAR_INPUT
		ipContour	:	ITcVnContainer;	(* Source container with 2D points (TcVnPoint2_DINT or TcVnPoint2_REAL or TcVnPoint2_LREAL) *)
		eDirection	:	ETcVnExtremePointDirection;	(* Selects the search direction for the extreme point *)
	END_VAR
	VAR_IN_OUT
		aExtremePoint	:	TcVnPoint2_LREAL;	(* Returns the extreme point of the contour, according to eDirection *)
	END_VAR
	VAR_INPUT
		hrPrev	:	HRESULT;	(* HRESULT indicating the result of previous operations (If SUCCEEDED(hrPrev) equals false, no operation is executed.) *)
	END_VAR

END_FUNCTION

// Functions/Contour Analysis/F_VN_ContourInertiaRatio

	{attribute 'TcIecLibraryType'}
	{attribute 'external_name' := 'F_VN_ContourInertiaRatio_GUID_2335F023_8AD3_B107_707F_3B5949D37FF3'}
	(* Computes the inertia ratio of a contour which reflects how a contour/shape is elongated (i.e. circle: 1.0, line: 0.0). *)
	FUNCTION F_VN_ContourInertiaRatio : HRESULT
	VAR_INPUT
		ipContour	:	ITcVnContainer;	(* Single contour (ContainerType_Vector_TcVnPoint2_DINT or ContainerType_Vector_TcVnPoint2_REAL; The elements of this container are the points of the contour.) *)
	END_VAR
	VAR_IN_OUT
		fInertiaRatio	:	LREAL;	(* Returns the inertia raio of the contour [0..1] *)
	END_VAR
	VAR_INPUT
		hrPrev	:	HRESULT;	(* HRESULT indicating the result of previous operations (If SUCCEEDED(hrPrev) equals false, no operation is executed.) *)
	END_VAR

END_FUNCTION

// Functions/Contour Analysis/F_VN_ContourMoments

	{attribute 'TcIecLibraryType'}
	{attribute 'external_name' := 'F_VN_ContourMoments_GUID_4E317C39_BCD2_B97C_66FE_7B2E6184683C'}
	(* Computes the spatial moments, the central moments, and the central normalized moments of a contour up to the third order. *)
	FUNCTION F_VN_ContourMoments : HRESULT
	VAR_INPUT
		ipContour	:	ITcVnContainer;	(* Single contour (ContainerType_Vector_TcVnPoint2_DINT or ContainerType_Vector_TcVnPoint2_REAL; The elements of this container are the points of the contour.) *)
	END_VAR
	VAR_IN_OUT
		stMoments	:	TcVnMoments;	(* Returns a struct containing the moments *)
	END_VAR
	VAR_INPUT
		hrPrev	:	HRESULT;	(* HRESULT indicating the result of previous operations (If SUCCEEDED(hrPrev) equals false, no operation is executed.) *)
	END_VAR

END_FUNCTION

// Functions/Contour Analysis/F_VN_ContourOrientation

	{attribute 'TcIecLibraryType'}
	{attribute 'external_name' := 'F_VN_ContourOrientation_GUID_3A361B59_D61F_BB1C_51D1_3ECAC6644C4C'}
	(* Calculate the orientation of a contour or a set of points. *)
	FUNCTION F_VN_ContourOrientation : HRESULT
	VAR_INPUT
		ipContour	:	ITcVnContainer;	(* Source point set (ContainerType_Vector_TcVnPoint2_DINT, ContainerType_Vector_TcVnPoint2_REAL, or ContainerType_Vector_TcVnPoint2_LREAL. The elements of this container are the individual points.) *)
	END_VAR
	VAR_IN_OUT
		stOrientation	:	TcVnRotatedRectangle;	(* Resulting rotated rectangle, containig center of mass, lenghts of axes, and rotation angle of the contour in clockwise direction. *)
	END_VAR
	VAR_INPUT
		hrPrev	:	HRESULT;	(* HRESULT indicating the result of previous operations (If SUCCEEDED(hrPrev) equals false, no operation is executed.) *)
	END_VAR

END_FUNCTION

// Functions/Contour Analysis/F_VN_ContourOrientationExp

	{attribute 'TcIecLibraryType'}
	{attribute 'external_name' := 'F_VN_ContourOrientationExp_GUID_EE16A408_16A0_B98C_7F4E_C0EA2BD579F4'}
	(* Calculate the orientation of a contour or a set of points. (expert function) *)
	FUNCTION F_VN_ContourOrientationExp : HRESULT
	VAR_INPUT
		ipContour	:	ITcVnContainer;	(* Source point set (ContainerType_Vector_TcVnPoint2_DINT, ContainerType_Vector_TcVnPoint2_REAL, or ContainerType_Vector_TcVnPoint2_LREAL. The elements of this container are the individual points.) *)
	END_VAR
	VAR_IN_OUT
		stOrientation	:	TcVnRotatedRectangle;	(* Resulting rotated rectangle, containig center of mass, lenghts of axes, and rotation angle of the contour in clockwise direction. *)
	END_VAR
	VAR_INPUT
		eMethod	:	ETcVnOrientationMethod;	(* Method for calculating the orientation.  *)
		hrPrev	:	HRESULT;	(* HRESULT indicating the result of previous operations (If SUCCEEDED(hrPrev) equals false, no operation is executed.) *)
	END_VAR

END_FUNCTION

// Functions/Contour Analysis/F_VN_ContourPerimeter

	{attribute 'TcIecLibraryType'}
	{attribute 'external_name' := 'F_VN_ContourPerimeter_GUID_7EAA746C_3451_BDB1_6219_BA570A66CF5B'}
	(* Computes the perimeter of a contour (curve length if the contour is not closed). *)
	FUNCTION F_VN_ContourPerimeter : HRESULT
	VAR_INPUT
		ipContour	:	ITcVnContainer;	(* Single contour (ContainerType_Vector_TcVnPoint2_DINT or ContainerType_Vector_TcVnPoint2_REAL; The elements of this container are the points of the contour.) *)
	END_VAR
	VAR_IN_OUT
		fPerimeter	:	LREAL;	(* Returns the perimeter of the contour *)
	END_VAR
	VAR_INPUT
		bClosed	:	BOOL;	(* Specifys, if the contour is closed (first and last points connected) or not *)
		hrPrev	:	HRESULT;	(* HRESULT indicating the result of previous operations (If SUCCEEDED(hrPrev) equals false, no operation is executed.) *)
	END_VAR

END_FUNCTION

// Functions/Contour Analysis/F_VN_ContourRoundness

	{attribute 'TcIecLibraryType'}
	{attribute 'external_name' := 'F_VN_ContourRoundness_GUID_BDD94588_A606_B409_7C30_33D0F644472C'}
	(* Computes the roundness of a contour (perimeter^2 / area). *)
	FUNCTION F_VN_ContourRoundness : HRESULT
	VAR_INPUT
		ipContour	:	ITcVnContainer;	(* Single contour (ContainerType_Vector_TcVnPoint2_DINT or ContainerType_Vector_TcVnPoint2_REAL; The elements of this container are the points of the contour.) *)
	END_VAR
	VAR_IN_OUT
		fRoundness	:	LREAL;	(* Returns the roundness of the contour *)
	END_VAR
	VAR_INPUT
		hrPrev	:	HRESULT;	(* HRESULT indicating the result of previous operations (If SUCCEEDED(hrPrev) equals false, no operation is executed.) *)
	END_VAR

END_FUNCTION

// Functions/Contour Analysis/F_VN_ConvexHullPoints

	{attribute 'TcIecLibraryType'}
	{attribute 'external_name' := 'F_VN_ConvexHullPoints_GUID_E77E53A1_1151_B4F7_668C_B7BDD3CC4E38'}
	(* Determines the convex hull of a point set. *)
	FUNCTION F_VN_ConvexHullPoints : HRESULT
	VAR_INPUT
		ipPointSet	:	ITcVnContainer;	(* Source point set (ContainerType_Vector_TcVnPoint2_DINT or ContainerType_Vector_TcVnPoint2_REAL; The elements of this container are the individual points.) *)
		ipConvexHull	:	REFERENCE TO ITcVnContainer;	(* Returns a container which is filled with the sorted convex hull points (same type ID as ipPointSet; Non-zero interface pointers are reused.) *)
		hrPrev	:	HRESULT;	(* HRESULT indicating the result of previous operations (If SUCCEEDED(hrPrev) equals false, no operation is executed.) *)
	END_VAR

END_FUNCTION

// Functions/Contour Analysis/F_VN_ConvexHullPointsExp

	{attribute 'TcIecLibraryType'}
	{attribute 'external_name' := 'F_VN_ConvexHullPointsExp_GUID_AACE5CC3_4D27_B3A2_5916_32B3059A87D1'}
	(* Determines the convex hull of a point set. (expert function) *)
	FUNCTION F_VN_ConvexHullPointsExp : HRESULT
	VAR_INPUT
		ipPointSet	:	ITcVnContainer;	(* Source point set (ContainerType_Vector_TcVnPoint2_DINT or ContainerType_Vector_TcVnPoint2_REAL; The elements of this container are the individual points.) *)
		ipConvexHull	:	REFERENCE TO ITcVnContainer;	(* Returns a container which is filled with the sorted convex hull points (same type ID as ipPointSet; Non-zero interface pointers are reused.) *)
		bClockwise	:	BOOL;	(* Selects the sorting direction of the hull points, assuming cartesian coordinates. *)
		hrPrev	:	HRESULT;	(* HRESULT indicating the result of previous operations (If SUCCEEDED(hrPrev) equals false, no operation is executed.) *)
	END_VAR

END_FUNCTION

// Functions/Contour Analysis/F_VN_ConvexityDefects

	{attribute 'TcIecLibraryType'}
	{attribute 'external_name' := 'F_VN_ConvexityDefects_GUID_606C1A73_A6D1_B2E2_6D42_7D6F55AA8DB2'}
	(* Finds the convexity defects of a point set. *)
	FUNCTION F_VN_ConvexityDefects : HRESULT
	VAR_INPUT
		ipContour	:	ITcVnContainer;	(* Source contour (ContainerType_Vector_TcVnPoint2_DINT; The elements of this container are the individual points.) *)
		ipConvexityDefects	:	REFERENCE TO ITcVnContainer;	(* Returns a container which is filled with the convexity defects (ContainerType_Vector_TcVnVector4_DINT with [startIndex, endIndex, furthestPointIndex, fixedPointDistance (8 fraction bits, i.e. divide by 256 to get the distance in pixels)]; Non-zero interface pointers are reused.) *)
		hrPrev	:	HRESULT;	(* HRESULT indicating the result of previous operations (If SUCCEEDED(hrPrev) equals false, no operation is executed.) *)
	END_VAR

END_FUNCTION

// Functions/Contour Analysis/F_VN_CustomElementWiseContainerOperation_ITcVnContainer

	{attribute 'TcIecLibraryType'}
	{attribute 'external_name' := 'F_VN_CustomElementWiseContainerOperation_ITcVnContainer_GUID_3FA76E7B_9B7A_BC91_537C_68E8B7680611'}
	(* Performs a custom, element wise operation on a set of up to 3 containers. *)
	FUNCTION F_VN_CustomElementWiseContainerOperation_ITcVnContainer : HRESULT
	VAR_INPUT
		ipContainer1	:	ITcVnContainer;	(* Container 1 *)
		ipContainer2	:	ITcVnContainer;	(* Container 2 *)
		ipContainer3	:	ITcVnContainer;	(* Container 3 *)
		ipOperationFB	:	ITcVnCustomContainerOperation_ITcVnContainer;	(* Custom operation on the container elements *)
		hrPrev	:	HRESULT;	(* HRESULT indicating the result of previous operations (If SUCCEEDED(hrPrev) equals false, no operation is executed.) *)
	END_VAR

END_FUNCTION

// Interfaces/Containers/Function Blocks/ITcVnCustomContainerOperation_ITcVnContainer

	(* Offers an interface for custom, elementwise container operations (for containers of containers) with up to 3 different containers. *)
	{attribute 'c++_compatible'}
	INTERFACE ITcVnCustomContainerOperation_ITcVnContainer


(* Executes the custom operation on the container elements. *)
	{attribute 'c++_compatible'}
	{attribute 'minimal_input_size' := '4'}
	{attribute 'pack_mode' := '4'}
	METHOD Execute : HRESULT
	VAR_INPUT
		ipElement1 : ITcVnContainer;
		ipElement2 : ITcVnContainer;
		ipElement3 : ITcVnContainer;
	END_VAR
END_METHOD

END_INTERFACE

// Functions/Contour Analysis/F_VN_CustomElementWiseContainerOperation_ITcVnForwardIterator

	{attribute 'TcIecLibraryType'}
	{attribute 'external_name' := 'F_VN_CustomElementWiseContainerOperation_ITcVnForwardIterator_GUID_170D588C_FA8E_BC95_4489_48AE4B3EB2A8'}
	(* Performs a custom, element wise operation on a set of up to 3 containers. *)
	FUNCTION F_VN_CustomElementWiseContainerOperation_ITcVnForwardIterator : HRESULT
	VAR_INPUT
		ipContainer1	:	ITcVnContainer;	(* Container 1 *)
		ipContainer2	:	ITcVnContainer;	(* Container 2 *)
		ipContainer3	:	ITcVnContainer;	(* Container 3 *)
		ipOperationFB	:	ITcVnCustomContainerOperation_ITcVnForwardIterator;	(* Custom operation on the elements *)
		hrPrev	:	HRESULT;	(* HRESULT indicating the result of previous operations (If SUCCEEDED(hrPrev) equals false, no operation is executed.) *)
	END_VAR

END_FUNCTION

// Interfaces/Containers/Function Blocks/ITcVnCustomContainerOperation_ITcVnForwardIterator

	(* Offers an interface for custom, elementwise container operations with up to 3 different containers. *)
	{attribute 'c++_compatible'}
	INTERFACE ITcVnCustomContainerOperation_ITcVnForwardIterator


(* Executes the custom operation on the container elements. *)
	{attribute 'c++_compatible'}
	{attribute 'minimal_input_size' := '4'}
	{attribute 'pack_mode' := '4'}
	METHOD Execute : HRESULT
	VAR_INPUT
		ipElement1 : ITcVnForwardIterator;
		ipElement2 : ITcVnForwardIterator;
		ipElement3 : ITcVnForwardIterator;
	END_VAR
END_METHOD

END_INTERFACE

// Functions/Contour Analysis/F_VN_EnclosingCircle

	{attribute 'TcIecLibraryType'}
	{attribute 'external_name' := 'F_VN_EnclosingCircle_GUID_98B15731_BACD_B502_528B_7A9D14D2657D'}
	(* Searchs for a minimum area circle enclosing a set of points. *)
	FUNCTION F_VN_EnclosingCircle : HRESULT
	VAR_INPUT
		ipPointSet	:	ITcVnContainer;	(* Source point set (ContainerType_Vector_TcVnPoint2_DINT or ContainerType_Vector_TcVnPoint2_REAL; The elements of this container are the individual points.) *)
	END_VAR
	VAR_IN_OUT
		aCenter	:	TcVnPoint2_REAL;	(* Returns the center of the circle *)
		fRadius	:	REAL;	(* Returns the radius of the circle *)
	END_VAR
	VAR_INPUT
		hrPrev	:	HRESULT;	(* HRESULT indicating the result of previous operations (If SUCCEEDED(hrPrev) equals false, no operation is executed.) *)
	END_VAR

END_FUNCTION

// Functions/Contour Analysis/F_VN_EnclosingRectangle

	{attribute 'TcIecLibraryType'}
	{attribute 'external_name' := 'F_VN_EnclosingRectangle_GUID_EEE63742_1DDA_B16D_4ACD_5B6FBE1262FD'}
	(* Searches for a minimum area rectangle enclosing a set of points. *)
	FUNCTION F_VN_EnclosingRectangle : HRESULT
	VAR_INPUT
		ipPointSet	:	ITcVnContainer;	(* Source point set (ContainerType_Vector_TcVnPoint2_DINT or ContainerType_Vector_TcVnPoint2_REAL; The elements of this container are the individual points.) *)
	END_VAR
	VAR_IN_OUT
		stRectangle	:	TcVnRotatedRectangle;	(* Returns the determined rectangle *)
	END_VAR
	VAR_INPUT
		hrPrev	:	HRESULT;	(* HRESULT indicating the result of previous operations (If SUCCEEDED(hrPrev) equals false, no operation is executed.) *)
	END_VAR

END_FUNCTION

// Functions/Contour Analysis/F_VN_EnclosingTriangle

	{attribute 'TcIecLibraryType'}
	{attribute 'external_name' := 'F_VN_EnclosingTriangle_GUID_231A9D1C_C130_BF12_6F62_39E64CBAFB07'}
	(* Searches for a minimum area triangle enclosing a set of points. *)
	FUNCTION F_VN_EnclosingTriangle : HRESULT
	VAR_INPUT
		ipPointSet	:	ITcVnContainer;	(* Source point set (ContainerType_Vector_TcVnPoint2_DINT or ContainerType_Vector_TcVnPoint2_REAL; The elements of this container are the individual points.) *)
	END_VAR
	VAR_IN_OUT
		aTriangleVertices	:	TcVnArray3_Point2_REAL;	(* Returns the 3 triangle vertices *)
	END_VAR
	VAR_INPUT
		hrPrev	:	HRESULT;	(* HRESULT indicating the result of previous operations (If SUCCEEDED(hrPrev) equals false, no operation is executed.) *)
	END_VAR
	VAR_OUTPUT
		fArea	:	LREAL;	(* Returns the triangle area *)
	END_VAR

END_FUNCTION

// Functions/Contour Analysis/F_VN_FitEllipse

	{attribute 'TcIecLibraryType'}
	{attribute 'external_name' := 'F_VN_FitEllipse_GUID_25AEB453_4C1A_B5B0_53FF_D06022270B49'}
	(* Fit an ellipse in a point set. *)
	FUNCTION F_VN_FitEllipse : HRESULT
	VAR_INPUT
		ipPointSet	:	ITcVnContainer;	(* Source point set (ContainerType_Vector_TcVnPoint2_DINT or ContainerType_Vector_TcVnPoint2_REAL; At least 5 reasonable points are required! The elements of this container are the individual points.) *)
	END_VAR
	VAR_IN_OUT
		stEllipse	:	TcVnRotatedRectangle;	(* Resulting ellipse, described by a rotated rectangle. *)
	END_VAR
	VAR_INPUT
		hrPrev	:	HRESULT;	(* HRESULT indicating the result of previous operations (If SUCCEEDED(hrPrev) equals false, no operation is executed.) *)
	END_VAR

END_FUNCTION

// Functions/Contour Analysis/F_VN_FitLine

	{attribute 'TcIecLibraryType'}
	{attribute 'external_name' := 'F_VN_FitLine_GUID_05B80202_7F3C_BE87_7619_8B349001AAEC'}
	(* Fit a line into a point set. *)
	FUNCTION F_VN_FitLine : HRESULT
	VAR_INPUT
		ipPointSet	:	ITcVnContainer;	(* Source point set (ContainerType_Vector_TcVnPoint2_DINT or ContainerType_Vector_TcVnPoint2_REAL; The elements of this container are the individual points.) *)
	END_VAR
	VAR_IN_OUT
		aFitLine	:	TcVnVector4_LREAL;	(* Resulting line. The first and second element describe the x and y component of a vector collinear to the line. The third and fourth element describe the x and y component of a point on the line. *)
	END_VAR
	VAR_INPUT
		hrPrev	:	HRESULT;	(* HRESULT indicating the result of previous operations (If SUCCEEDED(hrPrev) equals false, no operation is executed.) *)
	END_VAR

END_FUNCTION

// Functions/Contour Analysis/F_VN_FitLineExp

	{attribute 'TcIecLibraryType'}
	{attribute 'external_name' := 'F_VN_FitLineExp_GUID_CD7307F8_5A17_B520_4EA5_452045EC1C98'}
	(* Fit a line into a point set. (expert function) *)
	FUNCTION F_VN_FitLineExp : HRESULT
	VAR_INPUT
		ipPointSet	:	ITcVnContainer;	(* Source point set (ContainerType_Vector_TcVnPoint2_DINT or ContainerType_Vector_TcVnPoint2_REAL; The elements of this container are the individual points.) *)
	END_VAR
	VAR_IN_OUT
		aFitLine	:	TcVnVector4_LREAL;	(* Resulting line. The first and second element describe the x and y component of a vector collinear to the line. The third and fourth element describe the x and y component of a point on the line. *)
	END_VAR
	VAR_INPUT
		eDistanceType	:	ETcVnDistanceType;	(* Distance computation method (supported: L1, L2, L12, FAIR, WELSCH, HUBER) *)
		fParam	:	LREAL;	(* Numerical parameter (c) for some eDistanceType (should be >= 0). If 0, an optimal value is chosen internally. *)
		fEpsRadius	:	LREAL;	(* Accuracy of the radius (distance of the line from the coordinate origin, should be > 0). A smaller value means higher accuracy. *)
		fEpsAngle	:	LREAL;	(* Accuracy of the angle (should be > 0). A smaller value means higher accuracy. *)
		hrPrev	:	HRESULT;	(* HRESULT indicating the result of previous operations (If SUCCEEDED(hrPrev) equals false, no operation is executed.) *)
	END_VAR

END_FUNCTION

// Functions/Contour Analysis/F_VN_FourierDescriptors

	{attribute 'TcIecLibraryType'}
	{attribute 'external_name' := 'F_VN_FourierDescriptors_GUID_9CC98047_FDCD_B8CE_6528_B148D0153D64'}
	(* Computes the fourier descriptors for a closed contour. *)
	FUNCTION F_VN_FourierDescriptors : HRESULT
	VAR_INPUT
		ipContour	:	ITcVnContainer;	(* Closed contour (ContainerType_Vector_TcVnPoint2_DINT or ContainerType_Vector_TcVnPoint2_REAL or ContainerType_Vector_TcVnPoint2_LREAL. Providing the full contour is strongly recommended, i.e. use TCVN_CAM_NONE for contour detection algorithms.) *)
		ipDescriptors	:	REFERENCE TO ITcVnContainer;	(* Returns the fourier descriptors for ipContour (Re0, Im0, Re1, Im1, ...; ContainerType_Vector_LREAL if ipContour is of type ContainerType_Vector_TcVnPoint2_LREAL, else ContainerType_Vector_REAL.) *)
		nDescriptors	:	DINT;	(* Specifies how many descriptors should be returned (set to -1 to return all computed descriptors, i.e. at least as many as the number of contour points) *)
		hrPrev	:	HRESULT;	(* HRESULT indicating the result of previous operations (If SUCCEEDED(hrPrev) equals false, no operation is executed.) *)
	END_VAR

END_FUNCTION

// Functions/Contour Analysis/F_VN_MatchContours

	{attribute 'TcIecLibraryType'}
	{attribute 'external_name' := 'F_VN_MatchContours_GUID_7342D2FB_3A2B_B9EC_6050_7242829AC8C1'}
	(* Compare contours using the Hu moment invariants. In case of multiple contours in each container, the best matches are found and the average dissimilarity over all matched contours is returned. *)
	FUNCTION F_VN_MatchContours : HRESULT
	VAR_INPUT
		ipContour1	:	ITcVnContainer;	(* First contour (ContainerType_Vector_TcVnPoint2_DINT or ContainerType_Vector_TcVnPoint2_REAL; The elements of this container are the points of the contour) or collection of multiple contours (ContainerType_Vector_Vector_TcVnPoint2_DINT) *)
		ipContour2	:	ITcVnContainer;	(* Second contour (same type as ipContour1) *)
		eComparisonMethod	:	ETcVnContoursMatchComparisonMethod;	(* Method used for comparing the Hu moment invariants of the contours *)
	END_VAR
	VAR_IN_OUT
		fDissimilarity	:	LREAL;	(* Returns the dissimilarity of the contours depending on the chosen comparison method *)
	END_VAR
	VAR_INPUT
		hrPrev	:	HRESULT;	(* HRESULT indicating the result of previous operations (If SUCCEEDED(hrPrev) equals false, no operation is executed.) *)
	END_VAR

END_FUNCTION

// Functions/Contour Analysis/F_VN_MatchContoursExp

	{attribute 'TcIecLibraryType'}
	{attribute 'external_name' := 'F_VN_MatchContoursExp_GUID_0239EB8F_35A7_B1F4_66B1_16D7A01600A6'}
	(* Compare contours using the Hu moment invariants (and optionally further aspects). In case of multiple contours in each container, the best matches are found and the average dissimilarity over all matched contours is returned. (expert function) *)
	FUNCTION F_VN_MatchContoursExp : HRESULT
	VAR_INPUT
		ipContour1	:	ITcVnContainer;	(* First contour (ContainerType_Vector_TcVnPoint2_DINT or ContainerType_Vector_TcVnPoint2_REAL; The elements of this container are the points of the contour) or collection of multiple contours (ContainerType_Vector_Vector_TcVnPoint2_DINT) *)
		ipContour2	:	ITcVnContainer;	(* Second contour (same type as ipContour1) *)
		eComparisonMethod	:	ETcVnContoursMatchComparisonMethod;	(* Method used for comparing the Hu moment invariants of the contours *)
	END_VAR
	VAR_IN_OUT
		fDissimilarity	:	LREAL;	(* Returns the dissimilarity of the contours depending on the chosen comparison method *)
	END_VAR
	VAR_INPUT
		fAreaFactor	:	LREAL;	(* If > 0, the relative area difference between contours is scaled by this factor and added to the computed dissimilarity *)
		fAbsPositionFactor	:	LREAL;	(* If > 0, the absolute position difference between contours (i.e. the coordinates of the geometric contour centers) is scaled by this factor and added to the computed dissimilarity *)
		fRelPositionFactor	:	LREAL;	(* If > 0, the relative position difference between contours is scaled by this factor and added to the computed dissimilarity (only used if matching multiple contours) *)
		fNumDiffFactor	:	LREAL;	(* If > 0, the difference between the number of contours in both containers is scaled by this factor and added to the computed dissimilarity (only used if matching multiple contours) *)
		hrPrev	:	HRESULT;	(* HRESULT indicating the result of previous operations (If SUCCEEDED(hrPrev) equals false, no operation is executed.) *)
	END_VAR

END_FUNCTION

// Functions/Contour Analysis/F_VN_MatchContours1vsN

	{attribute 'TcIecLibraryType'}
	{attribute 'external_name' := 'F_VN_MatchContours1vsN_GUID_CA747EE4_4AA4_B3C6_5788_910799F0A9E4'}
	(* Compare a reference contour with multiple other contours using the Hu moment invariants. Returns a sorted list of best matches. *)
	FUNCTION F_VN_MatchContours1vsN : HRESULT
	VAR_INPUT
		ipRefContour	:	ITcVnContainer;	(* Reference contour (ContainerType_Vector_TcVnPoint2_DINT or ContainerType_Vector_TcVnPoint2_REAL; The elements of this container are the points of the contour) *)
		ipContours	:	ITcVnContainer;	(* Collection of multiple contours (CTcVnContainer_Vector_Vector_TcVnPoint2_DINT) *)
		ipMatchIndexes	:	REFERENCE TO ITcVnContainer;	(* Returns the indexes of the best matches (CTcVnContainer_Vector_ULINT; sorted, first element is best match, i.e. has lowest dissimilarity) *)
		ipDissimilarities	:	REFERENCE TO ITcVnContainer;	(* Returns the computed dissimilarities of the best matches (CTcVnContainer_Vector_LREAL; Optional, set to 0 if not required; sorted corresponding to ipMatchIndexes) *)
		fDissimilarityThreshold	:	LREAL;	(* Neglect irrelevant matches, i.e. dissimilarity > fDissimilarityThreshold *)
		eComparisonMethod	:	ETcVnContoursMatchComparisonMethod;	(* Method used for comparing the Hu moment invariants of the contours *)
		hrPrev	:	HRESULT;	(* HRESULT indicating the result of previous operations (If SUCCEEDED(hrPrev) equals false, no operation is executed.) *)
	END_VAR

END_FUNCTION

// Functions/Contour Analysis/F_VN_MatchContours1vsNExp

	{attribute 'TcIecLibraryType'}
	{attribute 'external_name' := 'F_VN_MatchContours1vsNExp_GUID_87200201_C4FC_B8CF_678F_B51D0C7FA2A9'}
	(* Compare a reference contour with multiple other contours using the Hu moment invariants (and optionally further aspects). Returns a sorted list of best matches. (expert function) *)
	FUNCTION F_VN_MatchContours1vsNExp : HRESULT
	VAR_INPUT
		ipRefContour	:	ITcVnContainer;	(* Reference contour (ContainerType_Vector_TcVnPoint2_DINT or ContainerType_Vector_TcVnPoint2_REAL; The elements of this container are the points of the contour) *)
		ipContours	:	ITcVnContainer;	(* Collection of multiple contours (CTcVnContainer_Vector_Vector_TcVnPoint2_DINT) *)
		ipMatchIndexes	:	REFERENCE TO ITcVnContainer;	(* Returns the indexes of the best matches (CTcVnContainer_Vector_ULINT; sorted, first element is best match, i.e. has lowest dissimilarity) *)
		ipDissimilarities	:	REFERENCE TO ITcVnContainer;	(* Returns the computed dissimilarities of the best matches (CTcVnContainer_Vector_LREAL; Optional, set to 0 if not required; sorted corresponding to ipMatchIndexes) *)
		fDissimilarityThreshold	:	LREAL;	(* Neglect irrelevant matches, i.e. dissimilarity > fDissimilarityThreshold *)
		eComparisonMethod	:	ETcVnContoursMatchComparisonMethod;	(* Method used for comparing the Hu moment invariants of the contours *)
		fAreaFactor	:	LREAL;	(* If > 0, the relative area difference between contours is scaled by this factor and added to the computed dissimilarity *)
		fAbsPositionFactor	:	LREAL;	(* If > 0, the absolute position difference between contours (i.e. the coordinates of the geometric contour centers) is scaled by this factor and added to the computed dissimilarity *)
		hrPrev	:	HRESULT;	(* HRESULT indicating the result of previous operations (If SUCCEEDED(hrPrev) equals false, no operation is executed.) *)
	END_VAR

END_FUNCTION

// Functions/Contour Analysis/F_VN_UprightBoundingRectangle

	{attribute 'TcIecLibraryType'}
	{attribute 'external_name' := 'F_VN_UprightBoundingRectangle_GUID_C4D8F759_D68A_BE7A_7A07_4185CAB63208'}
	(* Determines the upright bounding rectangle of a set of points. *)
	FUNCTION F_VN_UprightBoundingRectangle : HRESULT
	VAR_INPUT
		ipPointSet	:	ITcVnContainer;	(* Source point set (ContainerType_Vector_TcVnPoint2_DINT or ContainerType_Vector_TcVnPoint2_REAL; The elements of this container are the individual points.) *)
	END_VAR
	VAR_IN_OUT
		stRectangle	:	TcVnRectangle_UDINT;	(* Returns the determined rectangle *)
	END_VAR
	VAR_INPUT
		hrPrev	:	HRESULT;	(* HRESULT indicating the result of previous operations (If SUCCEEDED(hrPrev) equals false, no operation is executed.) *)
	END_VAR

END_FUNCTION

// Functions/Image Filtering/F_VN_BilateralFilter

	{attribute 'TcIecLibraryType'}
	{attribute 'external_name' := 'F_VN_BilateralFilter_GUID_FF18FF35_6385_BF57_765D_ACC7830DD512'}
	(* Apply a Bilateral filter to smooth the image but preserve edges. *)
	FUNCTION F_VN_BilateralFilter : HRESULT
	VAR_INPUT
		ipSrcImage	:	ITcVnImage;	(* Source image *)
		ipDestImage	:	REFERENCE TO ITcVnImage;	(* Destination image (Must be different from ipSrcImage! An appropriate destination image will be created if required.) *)
		nDiameter	:	DINT;	(* Diameter of the pixel neighborhood used for filtering (e.g. 5, 7, 9). If <= 0, it is automatically chosen dependend on fSigmaSpace. *)
		fSigmaColor	:	LREAL;	(* Sigma used for color space filtering (> 0). A larger value means that farther colors are mixed together. *)
		fSigmaSpace	:	LREAL;	(* Sigma used for coordinate space filtering (> 0). A larger value means that farther pixels can influence each other. *)
		hrPrev	:	HRESULT;	(* HRESULT indicating the result of previous operations (If SUCCEEDED(hrPrev) equals false, no operation is executed.) *)
	END_VAR

END_FUNCTION

// Functions/Image Filtering/F_VN_BilateralFilterExp

	{attribute 'TcIecLibraryType'}
	{attribute 'external_name' := 'F_VN_BilateralFilterExp_GUID_03CEAAD9_EB61_B9F8_4F52_47373FC820D1'}
	(* Apply a Bilateral filter to smooth the image but preserve edges. (expert function) *)
	FUNCTION F_VN_BilateralFilterExp : HRESULT
	VAR_INPUT
		ipSrcImage	:	ITcVnImage;	(* Source image *)
		ipDestImage	:	REFERENCE TO ITcVnImage;	(* Destination image (Must be different from ipSrcImage! An appropriate destination image will be created if required.) *)
		nDiameter	:	DINT;	(* Diameter of the pixel neighborhood used for filtering (e.g. 5, 7, 9). If <= 0, it is automatically chosen dependend on fSigmaSpace. *)
		fSigmaColor	:	LREAL;	(* Sigma used for color space filtering (> 0). A larger value means that farther colors are mixed together. *)
		fSigmaSpace	:	LREAL;	(* Sigma used for coordinate space filtering (> 0). A larger value means that farther pixels can influence each other. *)
		eBorderType	:	ETcVnBorderInterpolationMethod;	(* Image border handling *)
		hrPrev	:	HRESULT;	(* HRESULT indicating the result of previous operations (If SUCCEEDED(hrPrev) equals false, no operation is executed.) *)
	END_VAR

END_FUNCTION

// Functions/Image Filtering/F_VN_BoxFilter

	{attribute 'TcIecLibraryType'}
	{attribute 'external_name' := 'F_VN_BoxFilter_GUID_383A78F9_353A_B4D2_70DC_B3FC292E0AE7'}
	(* Apply a box filter to an image. *)
	FUNCTION F_VN_BoxFilter : HRESULT
	VAR_INPUT
		ipSrcImage	:	ITcVnImage;	(* Source image *)
		ipDestImage	:	REFERENCE TO ITcVnImage;	(* Destination image (An appropriate destination image will be created if required.) *)
		nFilterWidth	:	UDINT;	(* Filter width in pixels *)
		nFilterHeight	:	UDINT;	(* Filter height in pixels *)
		hrPrev	:	HRESULT;	(* HRESULT indicating the result of previous operations (If SUCCEEDED(hrPrev) equals false, no operation is executed.) *)
	END_VAR

END_FUNCTION

// Functions/Image Filtering/F_VN_BoxFilterExp

	{attribute 'TcIecLibraryType'}
	{attribute 'external_name' := 'F_VN_BoxFilterExp_GUID_60989363_D64D_B3A6_5664_03F41A8C57DA'}
	(* Apply a box filter to an image. (expert function) *)
	FUNCTION F_VN_BoxFilterExp : HRESULT
	VAR_INPUT
		ipSrcImage	:	ITcVnImage;	(* Source image *)
		ipDestImage	:	REFERENCE TO ITcVnImage;	(* Destination image (An appropriate destination image will be created if required.) *)
		nFilterWidth	:	UDINT;	(* Filter width in pixels *)
		nFilterHeight	:	UDINT;	(* Filter height in pixels *)
		eDestDepth	:	ETcVnElementType;	(* Destination image depth *)
	END_VAR
	VAR_IN_OUT
		aAnchor	:	TcVnPoint;	(* Anchor point of the kernel ([-1, -1] for center) *)
	END_VAR
	VAR_INPUT
		bNormalize	:	BOOL;	(* If true, the kernel is normalized by nFilterWidth * nFilterHeight *)
		eBorderType	:	ETcVnBorderInterpolationMethod;	(* Image border handling *)
		hrPrev	:	HRESULT;	(* HRESULT indicating the result of previous operations (If SUCCEEDED(hrPrev) equals false, no operation is executed.) *)
	END_VAR

END_FUNCTION

// Functions/Image Filtering/F_VN_BrightBorderObjects

	{attribute 'TcIecLibraryType'}
	{attribute 'external_name' := 'F_VN_BrightBorderObjects_GUID_1E1771F5_43E2_BF31_6A0D_D991F4E01ADC'}
	(* Find bright objects connected to the image border within a gray-scale single-channel image. *)
	FUNCTION F_VN_BrightBorderObjects : HRESULT
	VAR_INPUT
		ipSrcImage	:	ITcVnImage;	(* Source image (USINT, UINT, INT, REAL, or LREAL, 1 channel) *)
		ipDestImage	:	REFERENCE TO ITcVnImage;	(* Destination image (An appropriate destination image will be created if required.) *)
		hrPrev	:	HRESULT;	(* HRESULT indicating the result of previous operations (If SUCCEEDED(hrPrev) equals false, no operation is executed.) *)
	END_VAR

END_FUNCTION

// Functions/Image Filtering/F_VN_CreateStructuringElement

	{attribute 'TcIecLibraryType'}
	{attribute 'external_name' := 'F_VN_CreateStructuringElement_GUID_3CCDA439_68A3_B4FD_52D2_37CDB3332848'}
	(* Creates a structuring element for the usage with morphological operators and allocate an appropriate data buffer. The initial reference count is set to one if a new image interface is created and kept, otherwise. *)
	FUNCTION F_VN_CreateStructuringElement : HRESULT
	VAR_INPUT
		ipStructuringElement	:	REFERENCE TO ITcVnImage;	(* Returns the created structuring element (Non-zero interface pointers are reused.) *)
		eShape	:	ETcVnStructuringElementShape;	(* Shape of the structuring element (rectangle, cross, or ellipse) *)
		nWidth	:	UDINT;	(* Width *)
		nHeight	:	UDINT;	(* Height *)
		hrPrev	:	HRESULT;	(* HRESULT indicating the result of previous operations (If SUCCEEDED(hrPrev) equals false, no operation is executed.) *)
	END_VAR

END_FUNCTION

// Functions/Image Filtering/F_VN_CustomFilter

	{attribute 'TcIecLibraryType'}
	{attribute 'external_name' := 'F_VN_CustomFilter_GUID_D880B6DA_1642_B4A6_7123_80876741FC17'}
	(* Apply a custom filter to the image. *)
	FUNCTION F_VN_CustomFilter : HRESULT
	VAR_INPUT
		ipSrcImage	:	ITcVnImage;	(* Source image *)
		ipDestImage	:	REFERENCE TO ITcVnImage;	(* Destination image (An appropriate destination image will be created if required.) *)
		eDestDepth	:	ETcVnElementType;	(* Destination image depth *)
	END_VAR
	VAR_IN_OUT
		stKernel	:	TcVnMatrix;	(* Custom filter kernel with values of type REAL or LREAL *)
	END_VAR
	VAR_INPUT
		hrPrev	:	HRESULT;	(* HRESULT indicating the result of previous operations (If SUCCEEDED(hrPrev) equals false, no operation is executed.) *)
	END_VAR

END_FUNCTION

// Functions/Image Filtering/F_VN_CustomFilterExp

	{attribute 'TcIecLibraryType'}
	{attribute 'external_name' := 'F_VN_CustomFilterExp_GUID_F097BF34_3128_B6C3_4676_31B039D16A85'}
	(* Apply a custom filter to the image. (expert function) *)
	FUNCTION F_VN_CustomFilterExp : HRESULT
	VAR_INPUT
		ipSrcImage	:	ITcVnImage;	(* Source image *)
		ipDestImage	:	REFERENCE TO ITcVnImage;	(* Destination image (An appropriate destination image will be created if required.) *)
		eDestDepth	:	ETcVnElementType;	(* Destination image depth *)
	END_VAR
	VAR_IN_OUT
		stKernel	:	TcVnMatrix;	(* Custom filter kernel with values of type REAL or LREAL *)
		aAnchor	:	TcVnPoint;	(* Anchor point of the kernel *)
	END_VAR
	VAR_INPUT
		fDelta	:	LREAL;	(* Value added to each pixel after filtering *)
		eBorderType	:	ETcVnBorderInterpolationMethod;	(* Image border handling *)
		hrPrev	:	HRESULT;	(* HRESULT indicating the result of previous operations (If SUCCEEDED(hrPrev) equals false, no operation is executed.) *)
	END_VAR

END_FUNCTION

// Functions/Image Filtering/F_VN_DarkBorderObjects

	{attribute 'TcIecLibraryType'}
	{attribute 'external_name' := 'F_VN_DarkBorderObjects_GUID_CBAB159C_9AE8_BFCA_6643_C2EA3A610492'}
	(* Find dark objects connected to the image border within a gray-scale single-channel image. (equivalent to filling holes) *)
	FUNCTION F_VN_DarkBorderObjects : HRESULT
	VAR_INPUT
		ipSrcImage	:	ITcVnImage;	(* Source image (USINT, UINT, INT, REAL, or LREAL, 1 channel) *)
		ipDestImage	:	REFERENCE TO ITcVnImage;	(* Destination image (An appropriate destination image will be created if required.) *)
		hrPrev	:	HRESULT;	(* HRESULT indicating the result of previous operations (If SUCCEEDED(hrPrev) equals false, no operation is executed.) *)
	END_VAR

END_FUNCTION

// Functions/Image Filtering/F_VN_FillHoles

	{attribute 'TcIecLibraryType'}
	{attribute 'external_name' := 'F_VN_FillHoles_GUID_AEDCB3CC_4399_B347_5E9A_30FC9F5A5EBC'}
	(* Fill holes within a gray-scale single-channel image. (equivalent to finding dark border objects) *)
	FUNCTION F_VN_FillHoles : HRESULT
	VAR_INPUT
		ipSrcImage	:	ITcVnImage;	(* Source image (USINT, UINT, INT, REAL, or LREAL, 1 channel) *)
		ipDestImage	:	REFERENCE TO ITcVnImage;	(* Destination image (An appropriate destination image will be created if required.) *)
		hrPrev	:	HRESULT;	(* HRESULT indicating the result of previous operations (If SUCCEEDED(hrPrev) equals false, no operation is executed.) *)
	END_VAR

END_FUNCTION

// Functions/Image Filtering/F_VN_GaussianFilter

	{attribute 'TcIecLibraryType'}
	{attribute 'external_name' := 'F_VN_GaussianFilter_GUID_7EB80A9C_6B07_BE4A_73B2_84F781E45325'}
	(* Apply a Gaussian filter to smooth the image. *)
	FUNCTION F_VN_GaussianFilter : HRESULT
	VAR_INPUT
		ipSrcImage	:	ITcVnImage;	(* Source image *)
		ipDestImage	:	REFERENCE TO ITcVnImage;	(* Destination image (An appropriate destination image will be created if required.) *)
		nFilterWidth	:	UDINT;	(* Filter width in pixels (1, 3, 5, 7, ...) *)
		nFilterHeight	:	UDINT;	(* Filter height in pixels (1, 3, 5, 7, ...) *)
		hrPrev	:	HRESULT;	(* HRESULT indicating the result of previous operations (If SUCCEEDED(hrPrev) equals false, no operation is executed.) *)
	END_VAR

END_FUNCTION

// Functions/Image Filtering/F_VN_GaussianFilterExp

	{attribute 'TcIecLibraryType'}
	{attribute 'external_name' := 'F_VN_GaussianFilterExp_GUID_AFB11C69_1780_BA03_70FF_F338D373F9DB'}
	(* Apply a Gaussian filter to smooth the image. (expert function) *)
	FUNCTION F_VN_GaussianFilterExp : HRESULT
	VAR_INPUT
		ipSrcImage	:	ITcVnImage;	(* Source image *)
		ipDestImage	:	REFERENCE TO ITcVnImage;	(* Destination image (An appropriate destination image will be created if required.) *)
		nFilterWidth	:	UDINT;	(* Filter width in pixels (1, 3, 5, 7, ...) *)
		nFilterHeight	:	UDINT;	(* Filter height in pixels (1, 3, 5, 7, ...) *)
		fSigmaX	:	LREAL;	(* Gaussian kernel standard deviation in X direction (>= 0, automatically chosen if 0) *)
		fSigmaY	:	LREAL;	(* Gaussian kernel standard deviation in Y direction (>= 0, automatically chosen if 0) *)
		eBorderType	:	ETcVnBorderInterpolationMethod;	(* Image border handling *)
		hrPrev	:	HRESULT;	(* HRESULT indicating the result of previous operations (If SUCCEEDED(hrPrev) equals false, no operation is executed.) *)
	END_VAR

END_FUNCTION

// Functions/Image Filtering/F_VN_LaplacianFilter

	{attribute 'TcIecLibraryType'}
	{attribute 'external_name' := 'F_VN_LaplacianFilter_GUID_C9E9DA9A_20DA_BAFC_486A_4CE8B7D3C0E6'}
	(* Apply a Laplacian filter to an image. *)
	FUNCTION F_VN_LaplacianFilter : HRESULT
	VAR_INPUT
		ipSrcImage	:	ITcVnImage;	(* Source image *)
		ipDestImage	:	REFERENCE TO ITcVnImage;	(* Destination image (An appropriate destination image will be created if required.) *)
		eDestDepth	:	ETcVnElementType;	(* Destination image depth *)
		hrPrev	:	HRESULT;	(* HRESULT indicating the result of previous operations (If SUCCEEDED(hrPrev) equals false, no operation is executed.) *)
	END_VAR

END_FUNCTION

// Functions/Image Filtering/F_VN_LaplacianFilterExp

	{attribute 'TcIecLibraryType'}
	{attribute 'external_name' := 'F_VN_LaplacianFilterExp_GUID_6BDF1527_6231_BFA0_4F7C_C0A5CB8A734B'}
	(* Apply a Laplacian filter to an image. (expert function) *)
	FUNCTION F_VN_LaplacianFilterExp : HRESULT
	VAR_INPUT
		ipSrcImage	:	ITcVnImage;	(* Source image *)
		ipDestImage	:	REFERENCE TO ITcVnImage;	(* Destination image (An appropriate destination image will be created if required.) *)
		eDestDepth	:	ETcVnElementType;	(* Destination image depth *)
		nKernelSize	:	UDINT;	(* Aperture size used to compute the second-derivative filters (1, 3, 5, ..., 31) *)
		fScale	:	LREAL;	(* Scale factor for the computed derivative values *)
		fDelta	:	LREAL;	(* Delta value that is added to the results before storing them *)
		eBorderType	:	ETcVnBorderInterpolationMethod;	(* Image border handling *)
		hrPrev	:	HRESULT;	(* HRESULT indicating the result of previous operations (If SUCCEEDED(hrPrev) equals false, no operation is executed.) *)
	END_VAR

END_FUNCTION

// Functions/Image Filtering/F_VN_LocalMaxima

	{attribute 'TcIecLibraryType'}
	{attribute 'external_name' := 'F_VN_LocalMaxima_GUID_E863FE3E_2A85_B7C2_7590_B54D8A8C2B5B'}
	(* Find local maxima in a gray-scale single-channel image. The found maxima are marked by a value of 1 in the destination image. *)
	FUNCTION F_VN_LocalMaxima : HRESULT
	VAR_INPUT
		ipSrcImage	:	ITcVnImage;	(* Source image (USINT or UINT, 1 channel) *)
		ipDestImage	:	REFERENCE TO ITcVnImage;	(* Destination image (Must be different from ipSrcImage! An appropriate destination image will be created if required.) *)
		hrPrev	:	HRESULT;	(* HRESULT indicating the result of previous operations (If SUCCEEDED(hrPrev) equals false, no operation is executed.) *)
	END_VAR

END_FUNCTION

// Functions/Image Filtering/F_VN_LocalMinima

	{attribute 'TcIecLibraryType'}
	{attribute 'external_name' := 'F_VN_LocalMinima_GUID_D83390A3_B107_BC52_655D_38585BC9EBB4'}
	(* Find local minima in a gray-scale single-channel image. The found minima are marked by a value of 1 in the destination image. *)
	FUNCTION F_VN_LocalMinima : HRESULT
	VAR_INPUT
		ipSrcImage	:	ITcVnImage;	(* Source image (USINT or UINT, 1 channel) *)
		ipDestImage	:	REFERENCE TO ITcVnImage;	(* Destination image (Must be different from ipSrcImage! An appropriate destination image will be created if required.) *)
		hrPrev	:	HRESULT;	(* HRESULT indicating the result of previous operations (If SUCCEEDED(hrPrev) equals false, no operation is executed.) *)
	END_VAR

END_FUNCTION

// Functions/Image Filtering/F_VN_MedianFilter

	{attribute 'TcIecLibraryType'}
	{attribute 'external_name' := 'F_VN_MedianFilter_GUID_F32081D8_2964_B7B2_7EFA_A789944182FC'}
	(* Apply a Median filter to an image. *)
	FUNCTION F_VN_MedianFilter : HRESULT
	VAR_INPUT
		ipSrcImage	:	ITcVnImage;	(* Source image (for nFilterSize 3 or 5: USINT, UINT, REAL. For bigger filters, only USINT is supported. *)
		ipDestImage	:	REFERENCE TO ITcVnImage;	(* Destination image (An appropriate destination image will be created if required.) *)
		nFilterSize	:	UDINT;	(* Size (width and height) of the filter (3, 5, 7, ...) *)
		hrPrev	:	HRESULT;	(* HRESULT indicating the result of previous operations (If SUCCEEDED(hrPrev) equals false, no operation is executed.) *)
	END_VAR

END_FUNCTION

// Functions/Image Filtering/F_VN_MorphologicalOperator

	{attribute 'TcIecLibraryType'}
	{attribute 'external_name' := 'F_VN_MorphologicalOperator_GUID_592B9DA8_4B35_BA60_5277_06CED122307B'}
	(* Apply a morphological operator. *)
	FUNCTION F_VN_MorphologicalOperator : HRESULT
	VAR_INPUT
		ipSrcImage	:	ITcVnImage;	(* Source image (only 1 channel supported for reconstruction operators) *)
		ipDestImage	:	REFERENCE TO ITcVnImage;	(* Destination image (An appropriate destination image will be created if required.) *)
		eOperator	:	ETcVnMorphologicalOperator;	(* Operator type *)
		ipStructuringElement	:	ITcVnImage;	(* Structuring element to be applied (Typically created via F_VN_CreateStructuringElement.) *)
		hrPrev	:	HRESULT;	(* HRESULT indicating the result of previous operations (If SUCCEEDED(hrPrev) equals false, no operation is executed.) *)
	END_VAR

END_FUNCTION

// Functions/Image Filtering/F_VN_RemoveLocalMaxima

	{attribute 'TcIecLibraryType'}
	{attribute 'external_name' := 'F_VN_RemoveLocalMaxima_GUID_88BA04CE_1E90_BF67_52C8_F485FD4A67DB'}
	(* Remove local maxima up to a given height from a gray-scale single-channel image. *)
	FUNCTION F_VN_RemoveLocalMaxima : HRESULT
	VAR_INPUT
		ipSrcImage	:	ITcVnImage;	(* Source image (USINT, UINT, INT, REAL, or LREAL, 1 channel) *)
		ipDestImage	:	REFERENCE TO ITcVnImage;	(* Destination image (An appropriate destination image will be created if required.) *)
		fHeight	:	LREAL;	(* Maximum height of the maxima to be removed (must be greater than 0) *)
		hrPrev	:	HRESULT;	(* HRESULT indicating the result of previous operations (If SUCCEEDED(hrPrev) equals false, no operation is executed.) *)
	END_VAR

END_FUNCTION

// Functions/Image Filtering/F_VN_RemoveLocalMinima

	{attribute 'TcIecLibraryType'}
	{attribute 'external_name' := 'F_VN_RemoveLocalMinima_GUID_3E15036D_7BE0_B4EF_6736_1711DD1030BB'}
	(* Remove local minima up to a given height from a gray-scale single-channel image. *)
	FUNCTION F_VN_RemoveLocalMinima : HRESULT
	VAR_INPUT
		ipSrcImage	:	ITcVnImage;	(* Source image (USINT, UINT, INT, REAL, or LREAL, 1 channel) *)
		ipDestImage	:	REFERENCE TO ITcVnImage;	(* Destination image (An appropriate destination image will be created if required.) *)
		fHeight	:	LREAL;	(* Maximum height of the minima to be removed (must be greater than 0) *)
		hrPrev	:	HRESULT;	(* HRESULT indicating the result of previous operations (If SUCCEEDED(hrPrev) equals false, no operation is executed.) *)
	END_VAR

END_FUNCTION

// Functions/Image Filtering/F_VN_ScharrFilter

	{attribute 'TcIecLibraryType'}
	{attribute 'external_name' := 'F_VN_ScharrFilter_GUID_A755E6CF_0665_B228_7C35_2061F6705C27'}
	(* Calculates the first order derivative in x or y direction using a Scharr filter. *)
	FUNCTION F_VN_ScharrFilter : HRESULT
	VAR_INPUT
		ipSrcImage	:	ITcVnImage;	(* Source image *)
		ipDestImage	:	REFERENCE TO ITcVnImage;	(* Destination image (An appropriate destination image will be created if required.) *)
		eDestDepth	:	ETcVnElementType;	(* Destination image depth *)
		eFilterDirection	:	ETcVnFilterDirection;	(* Filter direction *)
		hrPrev	:	HRESULT;	(* HRESULT indicating the result of previous operations (If SUCCEEDED(hrPrev) equals false, no operation is executed.) *)
	END_VAR

END_FUNCTION

// Functions/Image Filtering/F_VN_ScharrFilterExp

	{attribute 'TcIecLibraryType'}
	{attribute 'external_name' := 'F_VN_ScharrFilterExp_GUID_8F1704C9_6013_B9C1_783E_38206638DE0F'}
	(* Calculates the first order derivative in x or y direction using a Scharr filter. (expert function) *)
	FUNCTION F_VN_ScharrFilterExp : HRESULT
	VAR_INPUT
		ipSrcImage	:	ITcVnImage;	(* Source image *)
		ipDestImage	:	REFERENCE TO ITcVnImage;	(* Destination image (An appropriate destination image will be created if required.) *)
		eDestDepth	:	ETcVnElementType;	(* Destination image depth *)
		eFilterDirection	:	ETcVnFilterDirection;	(* Filter direction *)
		fScale	:	LREAL;	(* Scale factor for the computed derivative values *)
		fDelta	:	LREAL;	(* Delta value that is added to the results prior to storing them in dest *)
		eBorderType	:	ETcVnBorderInterpolationMethod;	(* Image border handling *)
		hrPrev	:	HRESULT;	(* HRESULT indicating the result of previous operations (If SUCCEEDED(hrPrev) equals false, no operation is executed.) *)
	END_VAR

END_FUNCTION

// Functions/Image Filtering/F_VN_SeparableCustomFilter

